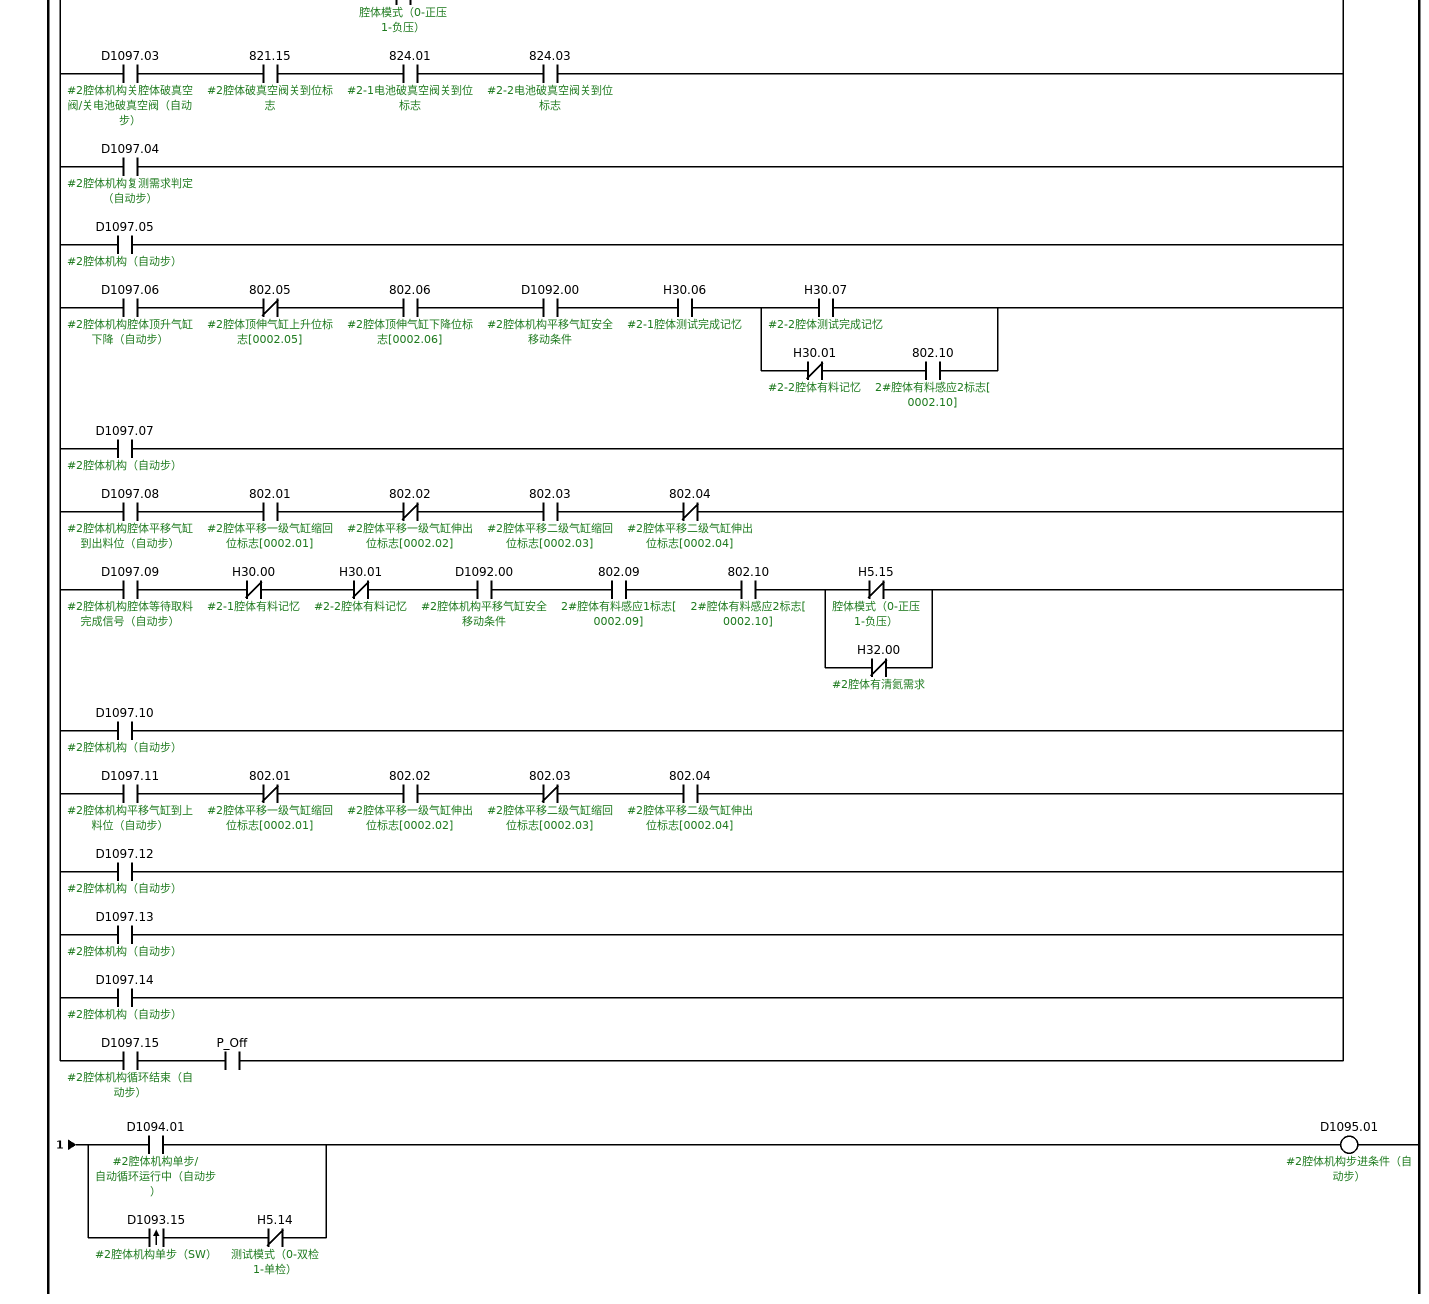
; [picture p264: 氦检机构 / 氦检腔2自动, rungs 7-7]
; rung 7: #2腔体机构步进条件（自动步）
LD D1096.00  ; #2腔体机构自动开始（自动步）
AND T1550  ; #2腔体机构开始运行条件延时(自动步)
LD D1096.01  ; #2腔体机构平移气缸到氦检位/数据初始化（自动步）
ANDNOT 802.01  ; #2腔体平移一级气缸缩回位标志[0002.01]
AND 802.02  ; #2腔体平移一级气缸伸出位标志[0002.02]
AND 802.03  ; #2腔体平移二级气缸缩回位标志[0002.03]
ANDNOT 802.04  ; #2腔体平移二级气缸伸出位标志[0002.04]
AND T1551  ; #2腔体机构数据初始化延时（自动步）
ORLD
LD D1096.02  ; #2腔体机构腔体顶升气缸上升（自动步）
AND 802.05  ; #2腔体顶伸气缸上升位标志[0002.05]
ANDNOT 802.06  ; #2腔体顶伸气缸下降位标志[0002.06]
ORLD
LD D1096.03  ; #2腔体机构等待氦检阀打开条件及腔体抽气阀打开条件/开腔体阀（自动步）
ANDNOT H27.00  ; #1腔体有清氦需求
LDNOT H37.00  ; #3腔体有清氦需求
ANDNOT H47.00  ; #4腔体有清氦需求
ANDNOT H57.00  ; 复检腔体有清氦需求
OR H6.02  ; 加速模式（1-开启）
ANDLD
AND D1092.15  ; #2腔体机构腔体抽气阀打开允许
AND D1092.14  ; #2腔体氦检阀打开允许条件
LD W380.15  ; 氦检仪漏率低于设定值（稳态）
OR H5.02  ; 氦检仪屏蔽
ANDLD
AND=L(301) D1104 #0  ; #2腔体机构清氦步序号
ORLD
OR D1096.04  ; #2腔体机构（自动步）
LD D1096.05  ; #2腔体机构腔体抽气阀打开/延时开电池抽气阀（自动步）
AND T2000  ; #2-1腔体抽真空阈值到达延时（测试）
ANDNOT H31.04  ; #2-1腔体抽真空NG
ANDNOT H31.05  ; #2-2腔体抽真空NG
LD 823.08  ; #2-1电池抽真空阀开到位标志
AND T2020  ; #2-1电池抽真空阈值到达延时（测试）
ANDNOT H31.00  ; #2-1电池泄漏
LD T2320  ; #2-2电池抽真空阈值到达延时（测试）
AND 823.10  ; #2-2电池抽真空阀开到位标志
ANDNOT H31.01  ; #2-2电池泄漏
ORNOT H30.01  ; #2-2腔体有料记忆
ANDLD
OR H5.15  ; 腔体模式（0-正压 1-负压）
OR H5.10  ; 空跑程序
ANDLD
ORLD
LD D1096.06  ; #2腔体机构关电池抽气阀（自动步）
ANDNOT W432.12  ; 设备氦气压力信号#1[alm]
ANDNOT W432.14  ; 设备注氦压力调节阀#1[alm]
AND 823.09  ; #2-1电池抽真空阀关到位标志
AND 823.11  ; #2-2电池抽真空阀关到位标志
ORLD
LD D1096.07  ; #2腔体机构开电池注氦阀（自动步）
LD 823.12  ; #2-1电池注氦阀开到位标志
AND T2024  ; #2-1电池注氦压力到达延时（测试）
LD 823.14  ; #2-2电池注氦阀开到位标志
AND T2324  ; #2-2电池注氦压力到达延时（测试）
ORNOT H30.01  ; #2-2腔体有料记忆
ANDLD
OR H31.02  ; #2-1电池注氦超时
OR H31.03  ; #2-2电池注氦超时
OR H5.15  ; 腔体模式（0-正压 1-负压）
OR H5.10  ; 空跑程序
ANDLD
ORLD
LD D1096.08  ; #2腔体机构关电池注氦阀（自动步）
AND 823.13  ; #2-1电池注氦阀关到位标志
AND 823.15  ; #2-2电池注氦阀关到位标志
ANDNOT H31.02  ; #2-1电池注氦超时
ANDNOT H31.03  ; #2-2电池注氦超时
LDNOT H31.08  ; #2-1注氦超限
ANDNOT H31.09  ; #2-2注氦超限
ORNOT H6.08  ; 注氦超限判断启用（1-启用）
ANDLD
ORLD
OR D1096.09  ; #2腔体机构（自动步）
LD D1096.10  ; #2腔体机构开腔体氦检阀/延时关腔体抽气阀（自动步）
LD T2006  ; #2-1腔体氦检数据取值判定延时（测试）
LD 820.10  ; 清氦保护阀1开到位标志[0000.10]
AND 802.07  ; #2腔体氦检阀开到位标志[0002.07]
OR H5.02  ; 氦检仪屏蔽
ANDLD
LD H31.06  ; #2-1腔体氦检时腔体压力过高
AND H31.07  ; #2-2腔体氦检时腔体压力过高
ORLD
ANDLD
ORLD
OR D1096.11  ; #2腔体机构（自动步）
LD D1096.12  ; #2腔体机构关腔体氦检阀（自动步）
AND 802.08  ; #2腔体氦检阀关到位标志[0002.08]
ANDNOT 802.07  ; #2腔体氦检阀开到位标志[0002.07]
LD 820.11  ; 清氦保护阀1阀关到位标志[0000.11]
ORNOT H6.07  ; 氦检完成后关闭氦检保护阀（1-氦检后关闭）
ANDLD
ORLD
OR D1096.13  ; #2腔体机构（自动步）
LD D1096.14  ; #2腔体机构开腔体#2-1腔体阀/开腔体#2-2腔体阀（自动步）
AND 802.08  ; #2腔体氦检阀关到位标志[0002.08]
ANDNOT H5.15  ; 腔体模式（0-正压 1-负压）
AND D1092.15  ; #2腔体机构腔体抽气阀打开允许
ORLD
LD D1096.15  ; #2腔体机构开腔体抽真空阀/开电池抽真空阀（自动步）
LD T2007  ; #2-1腔体抽残气压力到达延时（测试）
OR T2008  ; #2-1腔体抽残气时间上限到达延时（测试）
ANDLD
LD T2026  ; #2-1电池抽残气压力到达延时（测试）
OR T2027  ; #2-1电池抽残气时间上限到达延时（测试）
LD T2326  ; #2-2电池抽残气压力到达延时（测试）
OR T2327  ; #2-2电池抽残气时间上限到达延时（测试）
ANDLD
OR H5.10  ; 空跑程序
ANDLD
ORLD
LD D1097.00  ; #2腔体机构关腔体抽真空阀/关电池抽真空阀/开腔体阀（自动步）
AND 821.09  ; #2腔体抽真空阀关到位标志
AND 823.09  ; #2-1电池抽真空阀关到位标志
AND 823.11  ; #2-2电池抽真空阀关到位标志
ORLD
LD D1097.01  ; #2腔体机构清氦需求判定（自动步）
LDNOT H32.00  ; #2腔体有清氦需求
OR H5.15  ; 腔体模式（0-正压 1-负压）
ANDLD
ORLD
LD D1097.02  ; #2腔体机构开腔体破真空阀/开电池破真空阀（自动步）
AND T2002  ; #2-1腔体破真空阈值到达延时（测试）
LD T2022  ; #2-1电池破真空阈值到达延时（测试）
AND T2322  ; #2-2电池破真空阈值到达延时（测试）
OR H5.15  ; 腔体模式（0-正压 1-负压）
ANDLD
ORLD
LD D1097.03  ; #2腔体机构关腔体破真空阀/关电池破真空阀（自动步）
AND 821.15  ; #2腔体破真空阀关到位标志
AND 824.01  ; #2-1电池破真空阀关到位标志
AND 824.03  ; #2-2电池破真空阀关到位标志
ORLD
OR D1097.04  ; #2腔体机构复测需求判定（自动步）
OR D1097.05  ; #2腔体机构（自动步）
LD D1097.06  ; #2腔体机构腔体顶升气缸下降（自动步）
ANDNOT 802.05  ; #2腔体顶伸气缸上升位标志[0002.05]
AND 802.06  ; #2腔体顶伸气缸下降位标志[0002.06]
AND D1092.00  ; #2腔体机构平移气缸安全移动条件
AND H30.06  ; #2-1腔体测试完成记忆
LD H30.07  ; #2-2腔体测试完成记忆
LDNOT H30.01  ; #2-2腔体有料记忆
AND 802.10  ; 2#腔体有料感应2标志[0002.10]
ORLD
ANDLD
ORLD
OR D1097.07  ; #2腔体机构（自动步）
LD D1097.08  ; #2腔体机构腔体平移气缸到出料位（自动步）
AND 802.01  ; #2腔体平移一级气缸缩回位标志[0002.01]
ANDNOT 802.02  ; #2腔体平移一级气缸伸出位标志[0002.02]
AND 802.03  ; #2腔体平移二级气缸缩回位标志[0002.03]
ANDNOT 802.04  ; #2腔体平移二级气缸伸出位标志[0002.04]
ORLD
LD D1097.09  ; #2腔体机构腔体等待取料完成信号（自动步）  // 负压有清氦需求时，无需回初始位,直接跳回初始步序（D1096.00）
ANDNOT H30.00  ; #2-1腔体有料记忆
ANDNOT H30.01  ; #2-2腔体有料记忆
AND D1092.00  ; #2腔体机构平移气缸安全移动条件
AND 802.09  ; 2#腔体有料感应1标志[0002.09]
AND 802.10  ; 2#腔体有料感应2标志[0002.10]
LDNOT H5.15  ; 腔体模式（0-正压 1-负压）
ORNOT H32.00  ; #2腔体有清氦需求
ANDLD
ORLD
OR D1097.10  ; #2腔体机构（自动步）
LD D1097.11  ; #2腔体机构平移气缸到上料位（自动步）
ANDNOT 802.01  ; #2腔体平移一级气缸缩回位标志[0002.01]
AND 802.02  ; #2腔体平移一级气缸伸出位标志[0002.02]
ANDNOT 802.03  ; #2腔体平移二级气缸缩回位标志[0002.03]
AND 802.04  ; #2腔体平移二级气缸伸出位标志[0002.04]
ORLD
OR D1097.12  ; #2腔体机构（自动步）
OR D1097.13  ; #2腔体机构（自动步）
OR D1097.14  ; #2腔体机构（自动步）
LD D1097.15  ; #2腔体机构循环结束（自动步）
AND P_Off
ORLD
LD D1094.01  ; #2腔体机构单步/自动循环运行中（自动步）
@LD D1093.15  ; #2腔体机构单步（SW）
ANDNOT H5.14  ; 测试模式（0-双检 1-单检）
ORLD
ANDLD
OUT D1095.01  ; #2腔体机构步进条件（自动步）

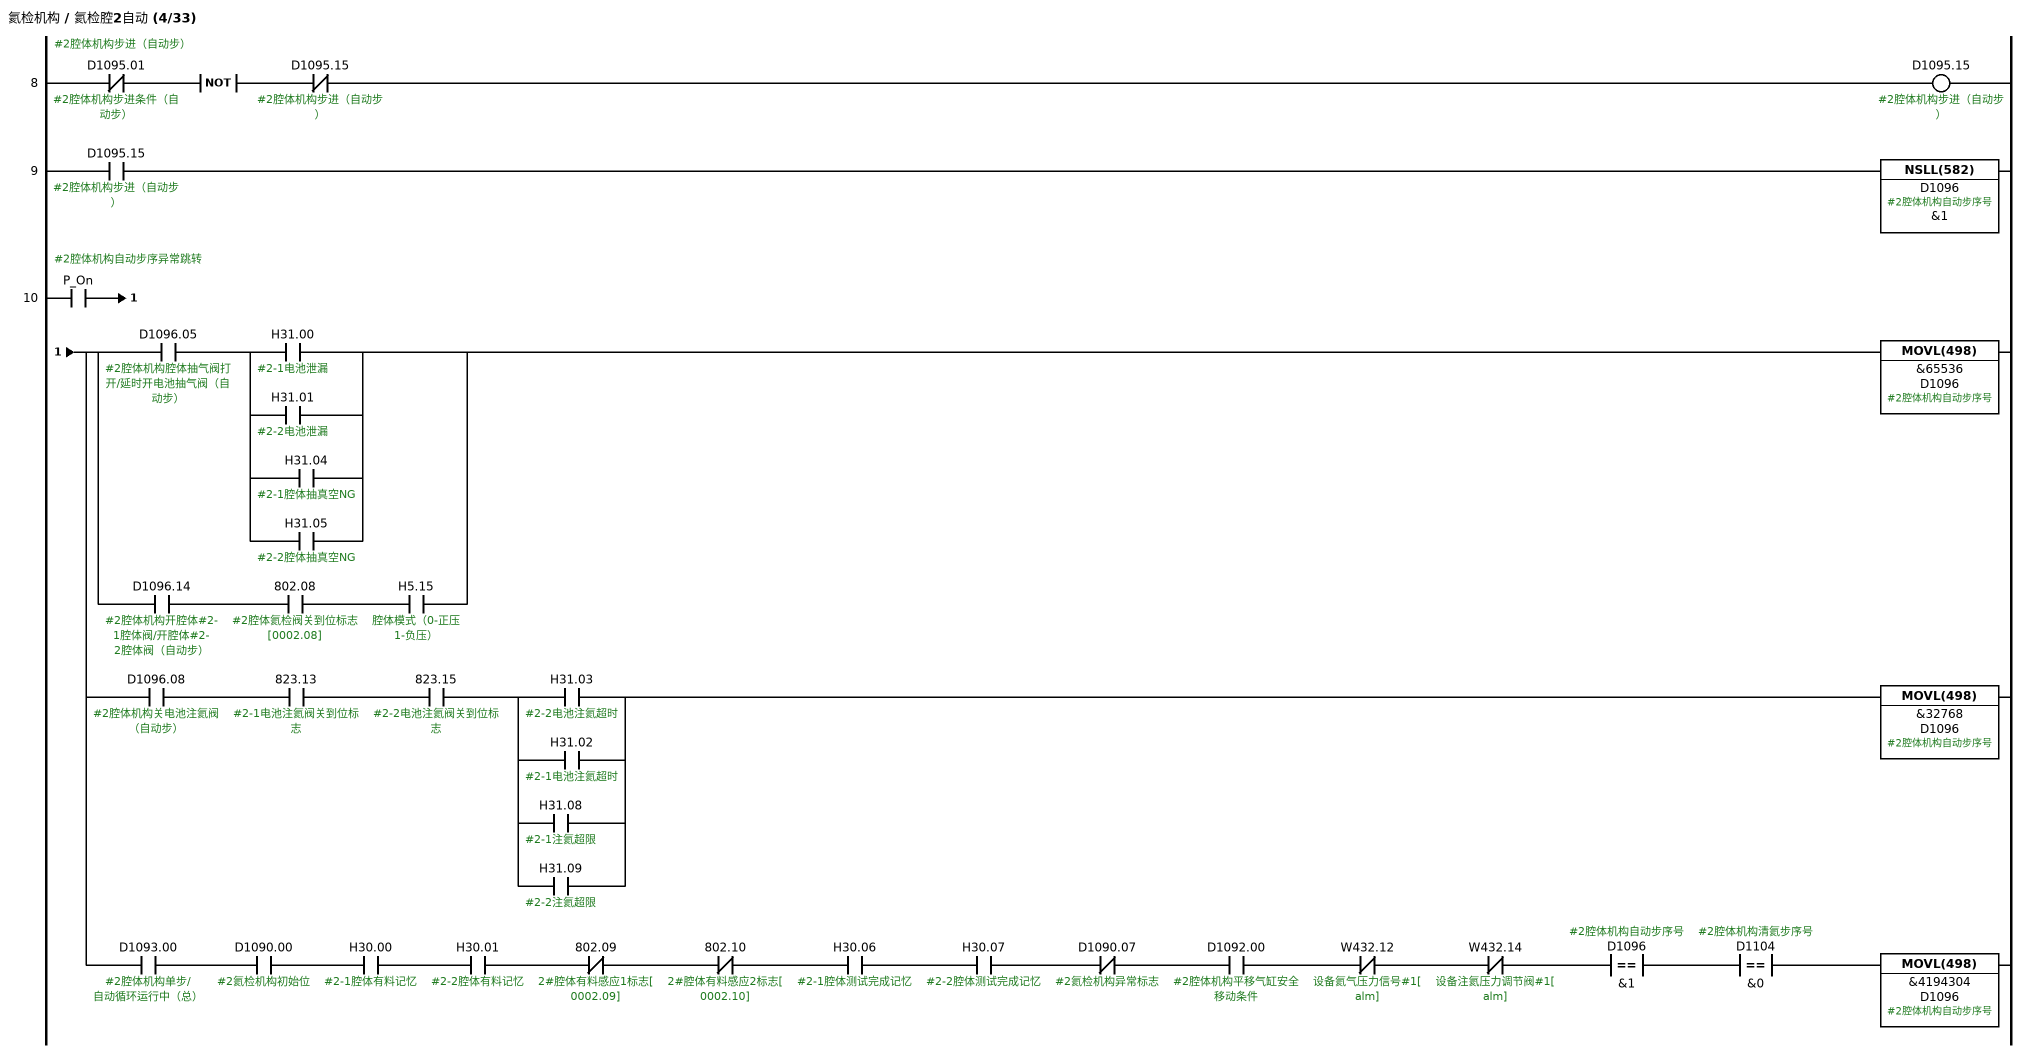
; rung 8: #2腔体机构步进（自动步）
LDNOT D1095.01  ; #2腔体机构步进条件（自动步）
NOT(520)
ANDNOT D1095.15  ; #2腔体机构步进（自动步）
OUT D1095.15  ; #2腔体机构步进（自动步）
; rung 9
LD D1095.15  ; #2腔体机构步进（自动步）
NSLL(582) D1096 &1  ; #2腔体机构自动步序号
; rung 10: #2腔体机构自动步序异常跳转
LD P_On
OUT TR0
LD D1096.05  ; #2腔体机构腔体抽气阀打开/延时开电池抽气阀（自动步）
LD H31.00  ; #2-1电池泄漏
OR H31.01  ; #2-2电池泄漏
OR H31.04  ; #2-1腔体抽真空NG
OR H31.05  ; #2-2腔体抽真空NG
ANDLD
LD D1096.14  ; #2腔体机构开腔体#2-1腔体阀/开腔体#2-2腔体阀（自动步）  // 负压模式不需要进行氦检后抽真空动作
AND 802.08  ; #2腔体氦检阀关到位标志[0002.08]
AND H5.15  ; 腔体模式（0-正压 1-负压）
ORLD
ANDLD
MOVL(498) &65536 D1096  ; #2腔体机构自动步序号  // 出现腔体抽真空NG，双电池抽真空NG，均跳转至自动步序D1067.0
LD TR0
AND D1096.08  ; #2腔体机构关电池注氦阀（自动步）
AND 823.13  ; #2-1电池注氦阀关到位标志
AND 823.15  ; #2-2电池注氦阀关到位标志
LD H31.03  ; #2-2电池注氦超时
OR H31.02  ; #2-1电池注氦超时
OR H31.08  ; #2-1注氦超限
OR H31.09  ; #2-2注氦超限
ANDLD
MOVL(498) &32768 D1096  ; #2腔体机构自动步序号
LD TR0
AND D1093.00  ; #2腔体机构单步/自动循环运行中（总）
AND D1090.00  ; #2氦检机构初始位
AND H30.00  ; #2-1腔体有料记忆
AND H30.01  ; #2-2腔体有料记忆
ANDNOT 802.09  ; 2#腔体有料感应1标志[0002.09]
ANDNOT 802.10  ; 2#腔体有料感应2标志[0002.10]
AND H30.06  ; #2-1腔体测试完成记忆
AND H30.07  ; #2-2腔体测试完成记忆
ANDNOT D1090.07  ; #2氦检机构异常标志
AND D1092.00  ; #2腔体机构平移气缸安全移动条件
ANDNOT W432.12  ; 设备氦气压力信号#1[alm]
ANDNOT W432.14  ; 设备注氦压力调节阀#1[alm]
AND=L(301) D1096 &1  ; #2腔体机构自动步序号
AND=L(301) D1104 &0  ; #2腔体机构清氦步序号
MOVL(498) &4194304 D1096  ; #2腔体机构自动步序号  // 带料复位，有测试完成物料跳转至D1097.06
; rung 11: ******************************* / 清氦步序 / *******************************

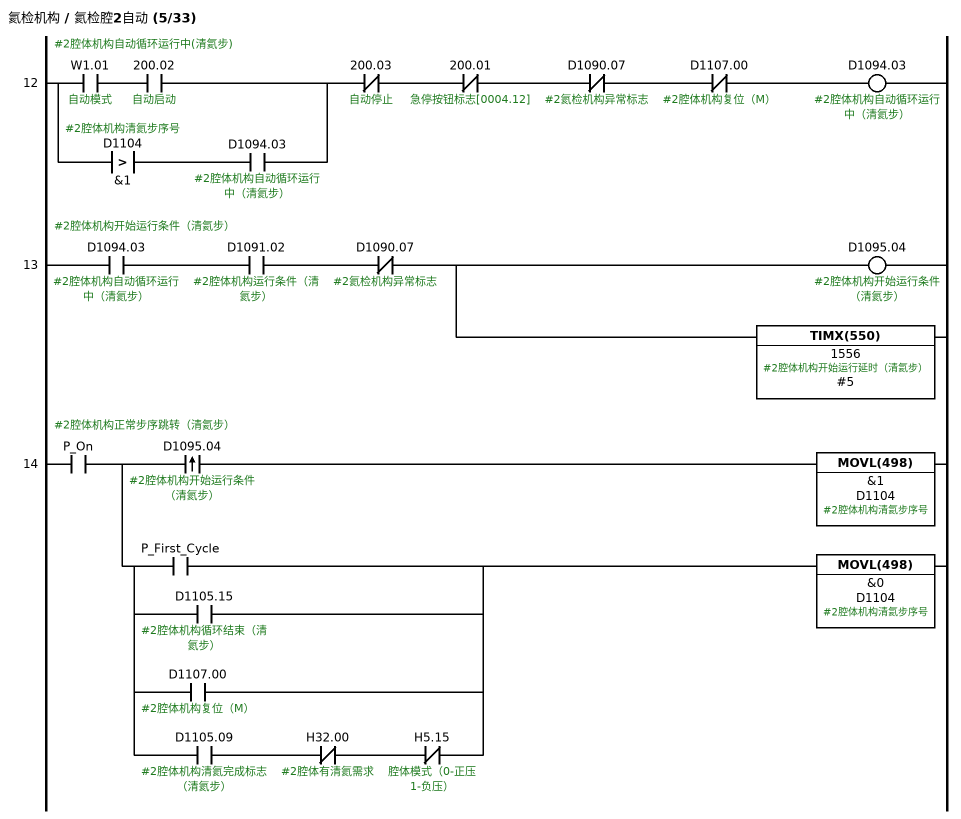
; rung 12: #2腔体机构自动循环运行中(清氦步)
LD W1.01  ; 自动模式
AND 200.02  ; 自动启动
LD>L(321) D1104 &1  ; #2腔体机构清氦步序号
AND D1094.03  ; #2腔体机构自动循环运行中（清氦步）
ORLD
ANDNOT 200.03  ; 自动停止
ANDNOT 200.01  ; 急停按钮标志[0004.12]
ANDNOT D1090.07  ; #2氦检机构异常标志
ANDNOT D1107.00  ; #2腔体机构复位（M）
OUT D1094.03  ; #2腔体机构自动循环运行中（清氦步）
; rung 13: #2腔体机构开始运行条件（清氦步）
LD D1094.03  ; #2腔体机构自动循环运行中（清氦步）
AND D1091.02  ; #2腔体机构运行条件（清氦步）
ANDNOT D1090.07  ; #2氦检机构异常标志
OUT D1095.04  ; #2腔体机构开始运行条件（清氦步）
TIMX(550) 1556 #5  ; #2腔体机构开始运行延时（清氦步）
; rung 14: #2腔体机构正常步序跳转（清氦步）
LD P_On
OUT TR0
@AND D1095.04  ; #2腔体机构开始运行条件（清氦步）
MOVL(498) &1 D1104  ; #2腔体机构清氦步序号
LD TR0
LD P_First_Cycle
OR D1105.15  ; #2腔体机构循环结束（清氦步）
OR D1107.00  ; #2腔体机构复位（M）
LD D1105.09  ; #2腔体机构清氦完成标志（清氦步）  // 正压腔体是待料清氦，需跳转回测试步序
ANDNOT H32.00  ; #2腔体有清氦需求
ANDNOT H5.15  ; 腔体模式（0-正压 1-负压）
ORLD
ANDLD
MOVL(498) &0 D1104  ; #2腔体机构清氦步序号

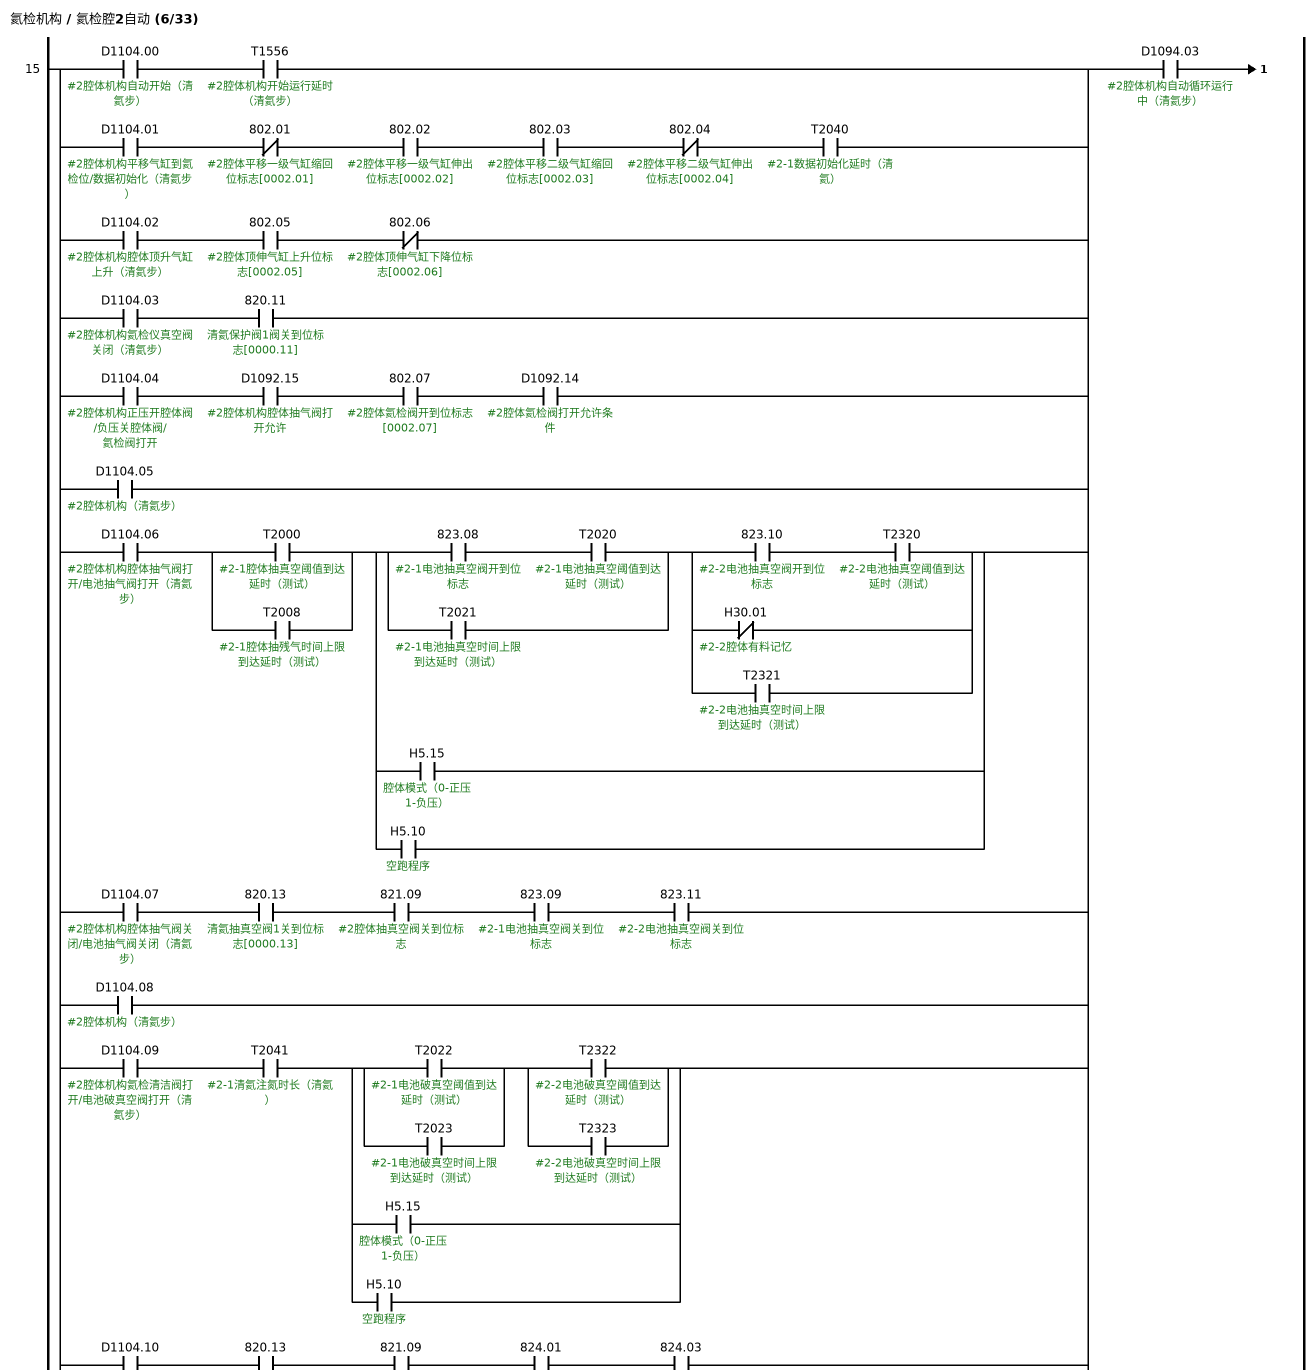

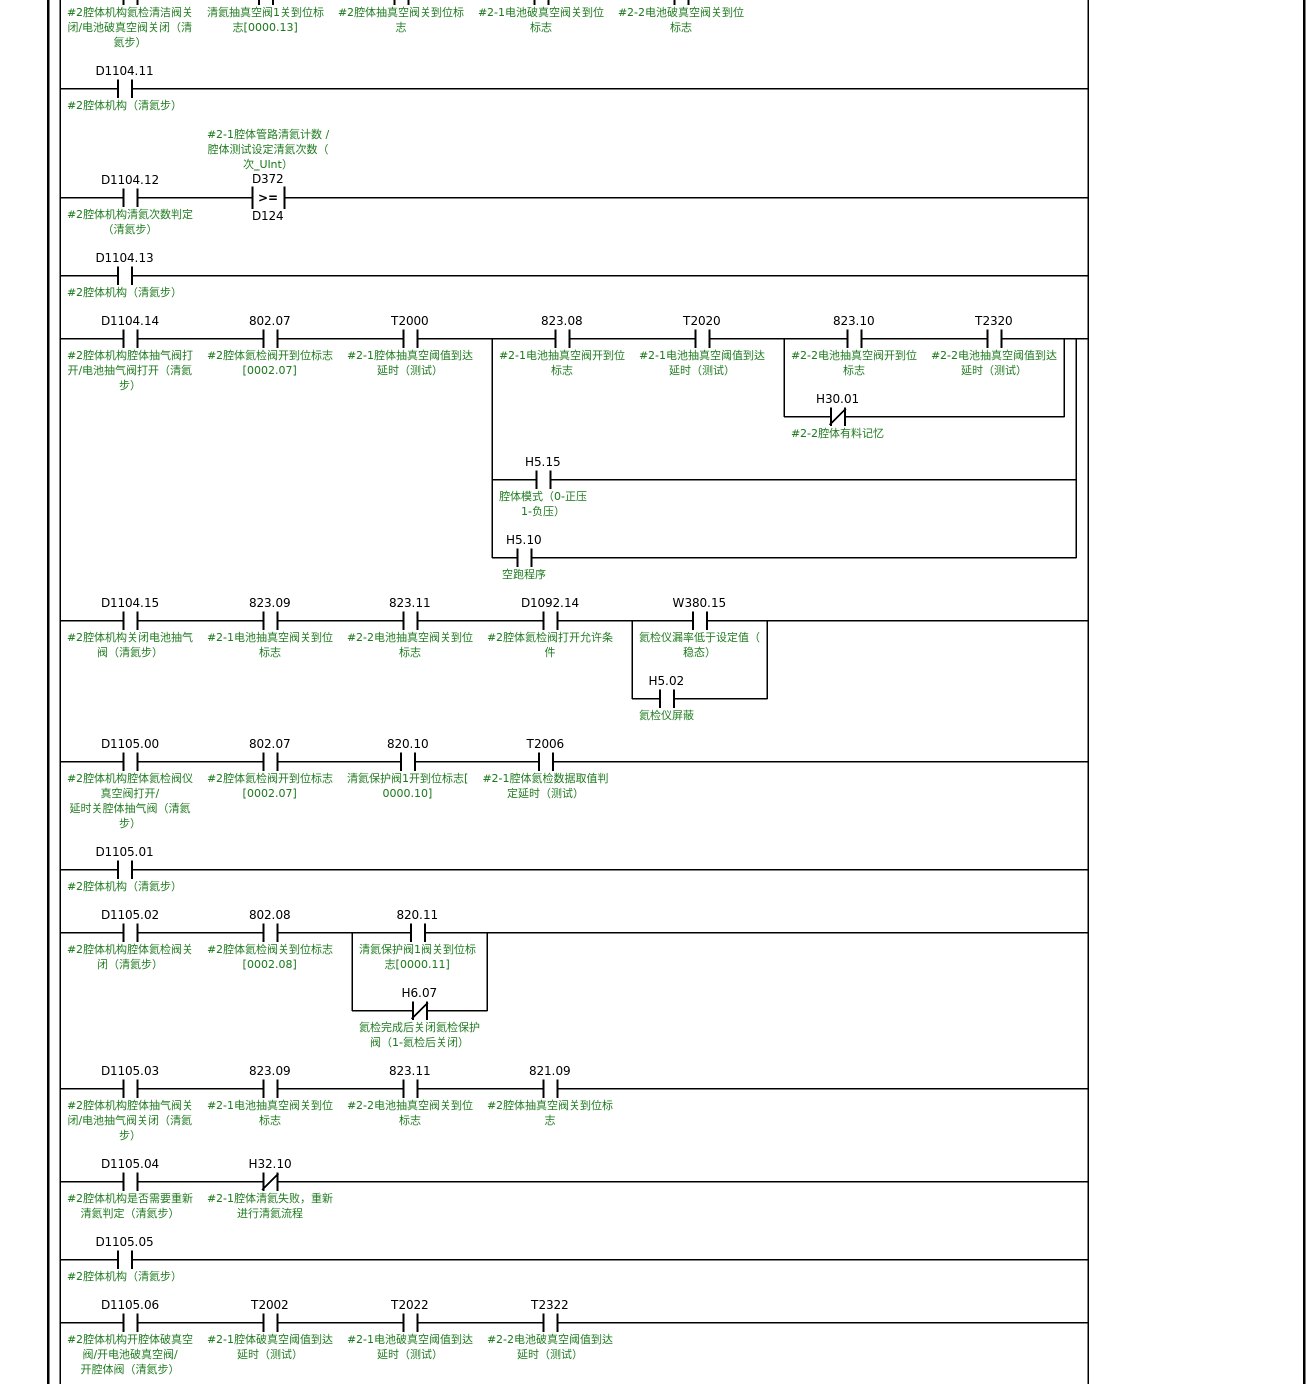

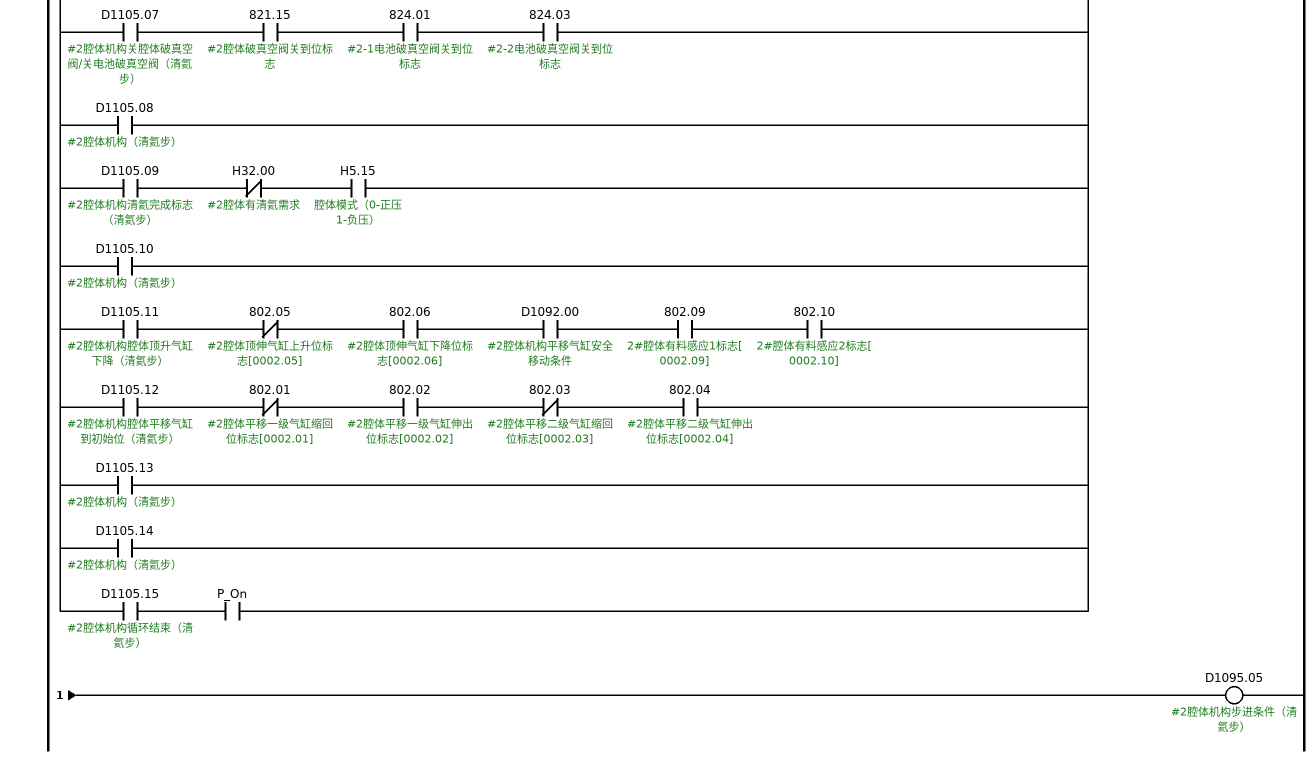
; rung 15
LD D1104.00  ; #2腔体机构自动开始（清氦步）
AND T1556  ; #2腔体机构开始运行延时（清氦步）
LD D1104.01  ; #2腔体机构平移气缸到氦检位/数据初始化（清氦步）
ANDNOT 802.01  ; #2腔体平移一级气缸缩回位标志[0002.01]
AND 802.02  ; #2腔体平移一级气缸伸出位标志[0002.02]
AND 802.03  ; #2腔体平移二级气缸缩回位标志[0002.03]
ANDNOT 802.04  ; #2腔体平移二级气缸伸出位标志[0002.04]
AND T2040  ; #2-1数据初始化延时（清氦）
ORLD
LD D1104.02  ; #2腔体机构腔体顶升气缸上升（清氦步）
AND 802.05  ; #2腔体顶伸气缸上升位标志[0002.05]
ANDNOT 802.06  ; #2腔体顶伸气缸下降位标志[0002.06]
ORLD
LD D1104.03  ; #2腔体机构氦检仪真空阀关闭（清氦步）
AND 820.11  ; 清氦保护阀1阀关到位标志[0000.11]
ORLD
LD D1104.04  ; #2腔体机构正压开腔体阀/负压关腔体阀/氦检阀打开  // 负压模式下，复测前的清氦不允许抽电池
AND D1092.15  ; #2腔体机构腔体抽气阀打开允许
AND 802.07  ; #2腔体氦检阀开到位标志[0002.07]
AND D1092.14  ; #2腔体氦检阀打开允许条件
ORLD
OR D1104.05  ; #2腔体机构（清氦步）
LD D1104.06  ; #2腔体机构腔体抽气阀打开/电池抽气阀打开（清氦步）
LD T2000  ; #2-1腔体抽真空阈值到达延时（测试）
OR T2008  ; #2-1腔体抽残气时间上限到达延时（测试）
ANDLD
LD 823.08  ; #2-1电池抽真空阀开到位标志
AND T2020  ; #2-1电池抽真空阈值到达延时（测试）
OR T2021  ; #2-1电池抽真空时间上限到达延时（测试）
LD 823.10  ; #2-2电池抽真空阀开到位标志
AND T2320  ; #2-2电池抽真空阈值到达延时（测试）
ORNOT H30.01  ; #2-2腔体有料记忆
OR T2321  ; #2-2电池抽真空时间上限到达延时（测试）
ANDLD
OR H5.15  ; 腔体模式（0-正压 1-负压）
OR H5.10  ; 空跑程序
ANDLD
ORLD
LD D1104.07  ; #2腔体机构腔体抽气阀关闭/电池抽气阀关闭（清氦步）
AND 820.13  ; 清氦抽真空阀1关到位标志[0000.13]
AND 821.09  ; #2腔体抽真空阀关到位标志
AND 823.09  ; #2-1电池抽真空阀关到位标志
AND 823.11  ; #2-2电池抽真空阀关到位标志
ORLD
OR D1104.08  ; #2腔体机构（清氦步）
LD D1104.09  ; #2腔体机构氦检清洁阀打开/电池破真空阀打开（清氦步）
AND T2041  ; #2-1清氦注氮时长（清氦）
LD T2022  ; #2-1电池破真空阈值到达延时（测试）
OR T2023  ; #2-1电池破真空时间上限到达延时（测试）
LD T2322  ; #2-2电池破真空阈值到达延时（测试）
OR T2323  ; #2-2电池破真空时间上限到达延时（测试）
ANDLD
OR H5.15  ; 腔体模式（0-正压 1-负压）
OR H5.10  ; 空跑程序
ANDLD
ORLD
LD D1104.10  ; #2腔体机构氦检清洁阀关闭/电池破真空阀关闭（清氦步）
AND 820.13  ; 清氦抽真空阀1关到位标志[0000.13]
AND 821.09  ; #2腔体抽真空阀关到位标志
AND 824.01  ; #2-1电池破真空阀关到位标志
AND 824.03  ; #2-2电池破真空阀关到位标志
ORLD
OR D1104.11  ; #2腔体机构（清氦步）
LD D1104.12  ; #2腔体机构清氦次数判定（清氦步）
AND>=(325) D372 D124  ; #2-1腔体管路清氦计数, 腔体测试设定清氦次数（次_UInt）
ORLD
OR D1104.13  ; #2腔体机构（清氦步）
LD D1104.14  ; #2腔体机构腔体抽气阀打开/电池抽气阀打开（清氦步）
AND 802.07  ; #2腔体氦检阀开到位标志[0002.07]
AND T2000  ; #2-1腔体抽真空阈值到达延时（测试）
LD 823.08  ; #2-1电池抽真空阀开到位标志
AND T2020  ; #2-1电池抽真空阈值到达延时（测试）
LD 823.10  ; #2-2电池抽真空阀开到位标志
AND T2320  ; #2-2电池抽真空阈值到达延时（测试）
ORNOT H30.01  ; #2-2腔体有料记忆
ANDLD
OR H5.15  ; 腔体模式（0-正压 1-负压）
OR H5.10  ; 空跑程序
ANDLD
ORLD
LD D1104.15  ; #2腔体机构关闭电池抽气阀（清氦步）
AND 823.09  ; #2-1电池抽真空阀关到位标志
AND 823.11  ; #2-2电池抽真空阀关到位标志
AND D1092.14  ; #2腔体氦检阀打开允许条件
LD W380.15  ; 氦检仪漏率低于设定值（稳态）
OR H5.02  ; 氦检仪屏蔽
ANDLD
ORLD
LD D1105.00  ; #2腔体机构腔体氦检阀仪真空阀打开/延时关腔体抽气阀（清氦步）
AND 802.07  ; #2腔体氦检阀开到位标志[0002.07]
AND 820.10  ; 清氦保护阀1开到位标志[0000.10]
AND T2006  ; #2-1腔体氦检数据取值判定延时（测试）
ORLD
OR D1105.01  ; #2腔体机构（清氦步）
LD D1105.02  ; #2腔体机构腔体氦检阀关闭（清氦步）
AND 802.08  ; #2腔体氦检阀关到位标志[0002.08]
LD 820.11  ; 清氦保护阀1阀关到位标志[0000.11]
ORNOT H6.07  ; 氦检完成后关闭氦检保护阀（1-氦检后关闭）
ANDLD
ORLD
LD D1105.03  ; #2腔体机构腔体抽气阀关闭/电池抽气阀关闭（清氦步）
AND 823.09  ; #2-1电池抽真空阀关到位标志
AND 823.11  ; #2-2电池抽真空阀关到位标志
AND 821.09  ; #2腔体抽真空阀关到位标志
ORLD
LD D1105.04  ; #2腔体机构是否需要重新清氦判定（清氦步）
ANDNOT H32.10  ; #2-1腔体清氦失败，重新进行清氦流程  // 清氦失败，重新进行清氦
ORLD
OR D1105.05  ; #2腔体机构（清氦步）
LD D1105.06  ; #2腔体机构开腔体破真空阀/开电池破真空阀/开腔体阀（清氦步）
AND T2002  ; #2-1腔体破真空阈值到达延时（测试）
AND T2022  ; #2-1电池破真空阈值到达延时（测试）
AND T2322  ; #2-2电池破真空阈值到达延时（测试）
ORLD
LD D1105.07  ; #2腔体机构关腔体破真空阀/关电池破真空阀（清氦步）
AND 821.15  ; #2腔体破真空阀关到位标志
AND 824.01  ; #2-1电池破真空阀关到位标志
AND 824.03  ; #2-2电池破真空阀关到位标志
ORLD
OR D1105.08  ; #2腔体机构（清氦步）
LD D1105.09  ; #2腔体机构清氦完成标志（清氦步）  // 正压腔体是待料清氦，需跳转回测试步序
ANDNOT H32.00  ; #2腔体有清氦需求
AND H5.15  ; 腔体模式（0-正压 1-负压）
ORLD
OR D1105.10  ; #2腔体机构（清氦步）
LD D1105.11  ; #2腔体机构腔体顶升气缸下降（清氦步）
ANDNOT 802.05  ; #2腔体顶伸气缸上升位标志[0002.05]
AND 802.06  ; #2腔体顶伸气缸下降位标志[0002.06]
AND D1092.00  ; #2腔体机构平移气缸安全移动条件
AND 802.09  ; 2#腔体有料感应1标志[0002.09]
AND 802.10  ; 2#腔体有料感应2标志[0002.10]
ORLD
LD D1105.12  ; #2腔体机构腔体平移气缸到初始位（清氦步）
ANDNOT 802.01  ; #2腔体平移一级气缸缩回位标志[0002.01]
AND 802.02  ; #2腔体平移一级气缸伸出位标志[0002.02]
ANDNOT 802.03  ; #2腔体平移二级气缸缩回位标志[0002.03]
AND 802.04  ; #2腔体平移二级气缸伸出位标志[0002.04]
ORLD
OR D1105.13  ; #2腔体机构（清氦步）
OR D1105.14  ; #2腔体机构（清氦步）
LD D1105.15  ; #2腔体机构循环结束（清氦步）
AND P_On
ORLD
AND D1094.03  ; #2腔体机构自动循环运行中（清氦步）
OUT D1095.05  ; #2腔体机构步进条件（清氦步）

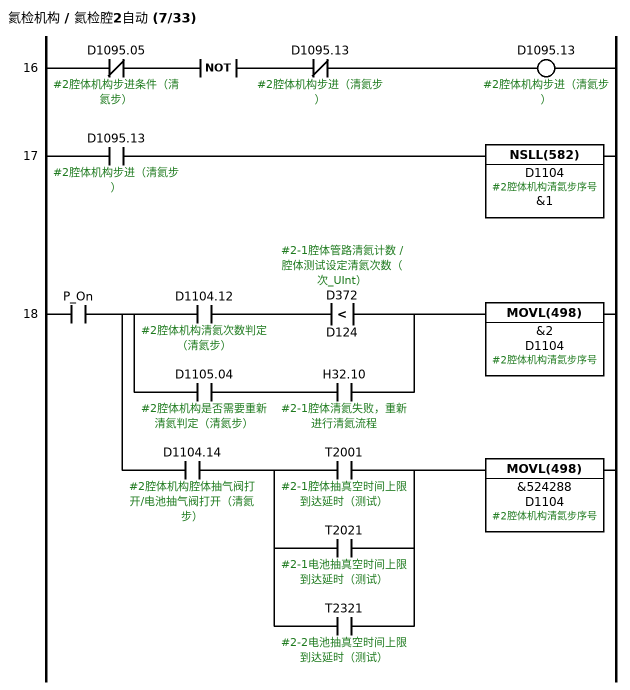
; rung 16
LDNOT D1095.05  ; #2腔体机构步进条件（清氦步）
NOT(520)
ANDNOT D1095.13  ; #2腔体机构步进（清氦步）
OUT D1095.13  ; #2腔体机构步进（清氦步）
; rung 17
LD D1095.13  ; #2腔体机构步进（清氦步）
NSLL(582) D1104 &1  ; #2腔体机构清氦步序号
; rung 18
LD P_On
OUT TR0
LD D1104.12  ; #2腔体机构清氦次数判定（清氦步）
AND<(310) D372 D124  ; #2-1腔体管路清氦计数, 腔体测试设定清氦次数（次_UInt）
LD D1105.04  ; #2腔体机构是否需要重新清氦判定（清氦步）
AND H32.10  ; #2-1腔体清氦失败，重新进行清氦流程  // 清氦失败，重新进行清氦
ORLD
ANDLD
MOVL(498) &2 D1104  ; #2腔体机构清氦步序号
LD TR0
AND D1104.14  ; #2腔体机构腔体抽气阀打开/电池抽气阀打开（清氦步）
LD T2001  ; #2-1腔体抽真空时间上限到达延时（测试）
OR T2021  ; #2-1电池抽真空时间上限到达延时（测试）
OR T2321  ; #2-2电池抽真空时间上限到达延时（测试）
ANDLD
MOVL(498) &524288 D1104  ; #2腔体机构清氦步序号  // 清氦过程腔体或电池抽气上限达到，均直接判定清氦完成，不进入氦检步序（跳转至D1075.03）

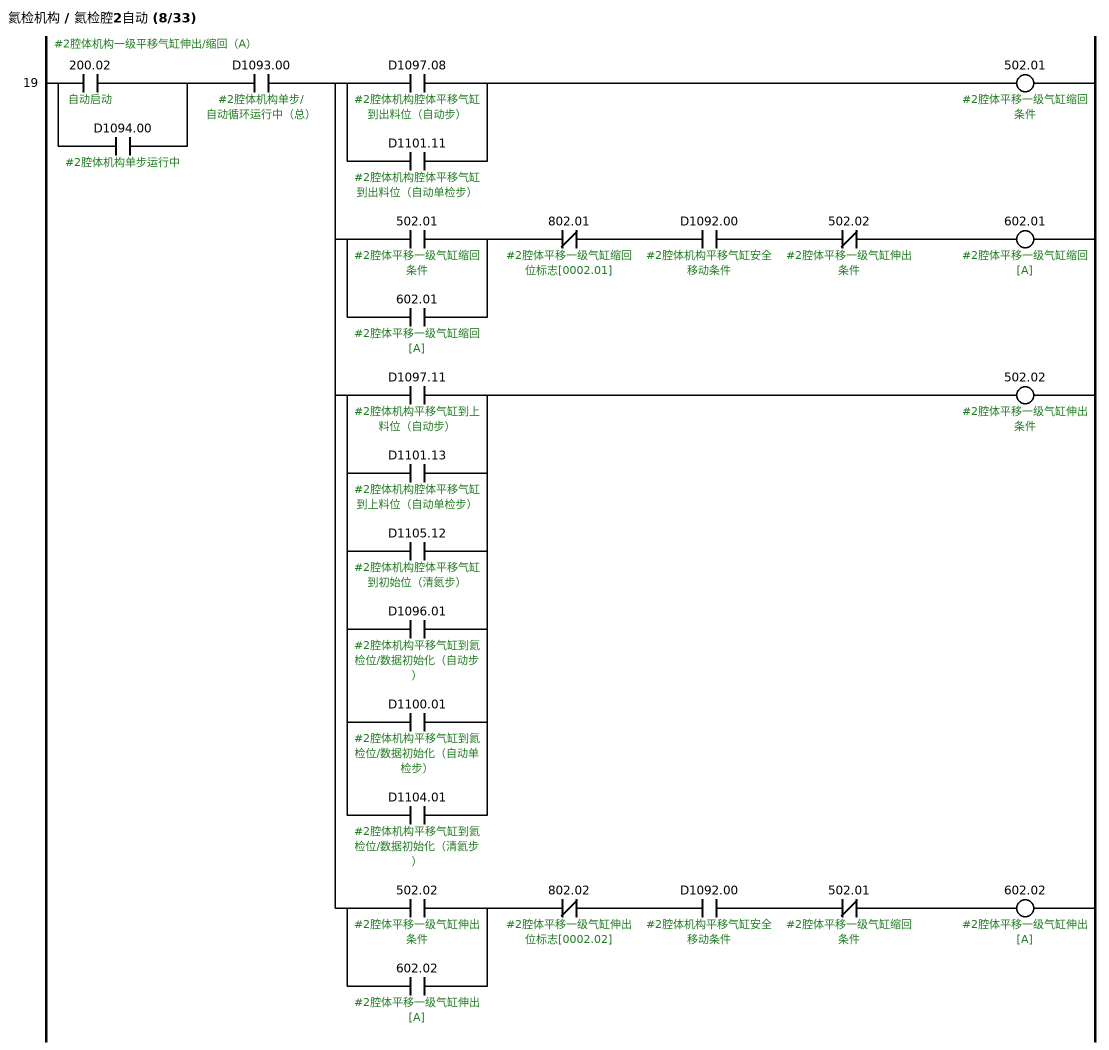
; rung 19: #2腔体机构一级平移气缸伸出/缩回（A）
LD 200.02  ; 自动启动
OR D1094.00  ; #2腔体机构单步运行中
AND D1093.00  ; #2腔体机构单步/自动循环运行中（总）
OUT TR0
LD D1097.08  ; #2腔体机构腔体平移气缸到出料位（自动步）
OR D1101.11  ; #2腔体机构腔体平移气缸到出料位（自动单检步）
ANDLD
OUT 502.01  ; #2腔体平移一级气缸缩回条件
LD TR0
LD 502.01  ; #2腔体平移一级气缸缩回条件
OR 602.01  ; #2腔体平移一级气缸缩回[A]
ANDLD
ANDNOT 802.01  ; #2腔体平移一级气缸缩回位标志[0002.01]
AND D1092.00  ; #2腔体机构平移气缸安全移动条件
ANDNOT 502.02  ; #2腔体平移一级气缸伸出条件
OUT 602.01  ; #2腔体平移一级气缸缩回[A]
LD TR0
LD D1097.11  ; #2腔体机构平移气缸到上料位（自动步）
OR D1101.13  ; #2腔体机构腔体平移气缸到上料位（自动单检步）
OR D1105.12  ; #2腔体机构腔体平移气缸到初始位（清氦步）
OR D1096.01  ; #2腔体机构平移气缸到氦检位/数据初始化（自动步）
OR D1100.01  ; #2腔体机构平移气缸到氦检位/数据初始化（自动单检步）
OR D1104.01  ; #2腔体机构平移气缸到氦检位/数据初始化（清氦步）
ANDLD
OUT 502.02  ; #2腔体平移一级气缸伸出条件
LD TR0
LD 502.02  ; #2腔体平移一级气缸伸出条件
OR 602.02  ; #2腔体平移一级气缸伸出[A]
ANDLD
ANDNOT 802.02  ; #2腔体平移一级气缸伸出位标志[0002.02]
AND D1092.00  ; #2腔体机构平移气缸安全移动条件
ANDNOT 502.01  ; #2腔体平移一级气缸缩回条件
OUT 602.02  ; #2腔体平移一级气缸伸出[A]

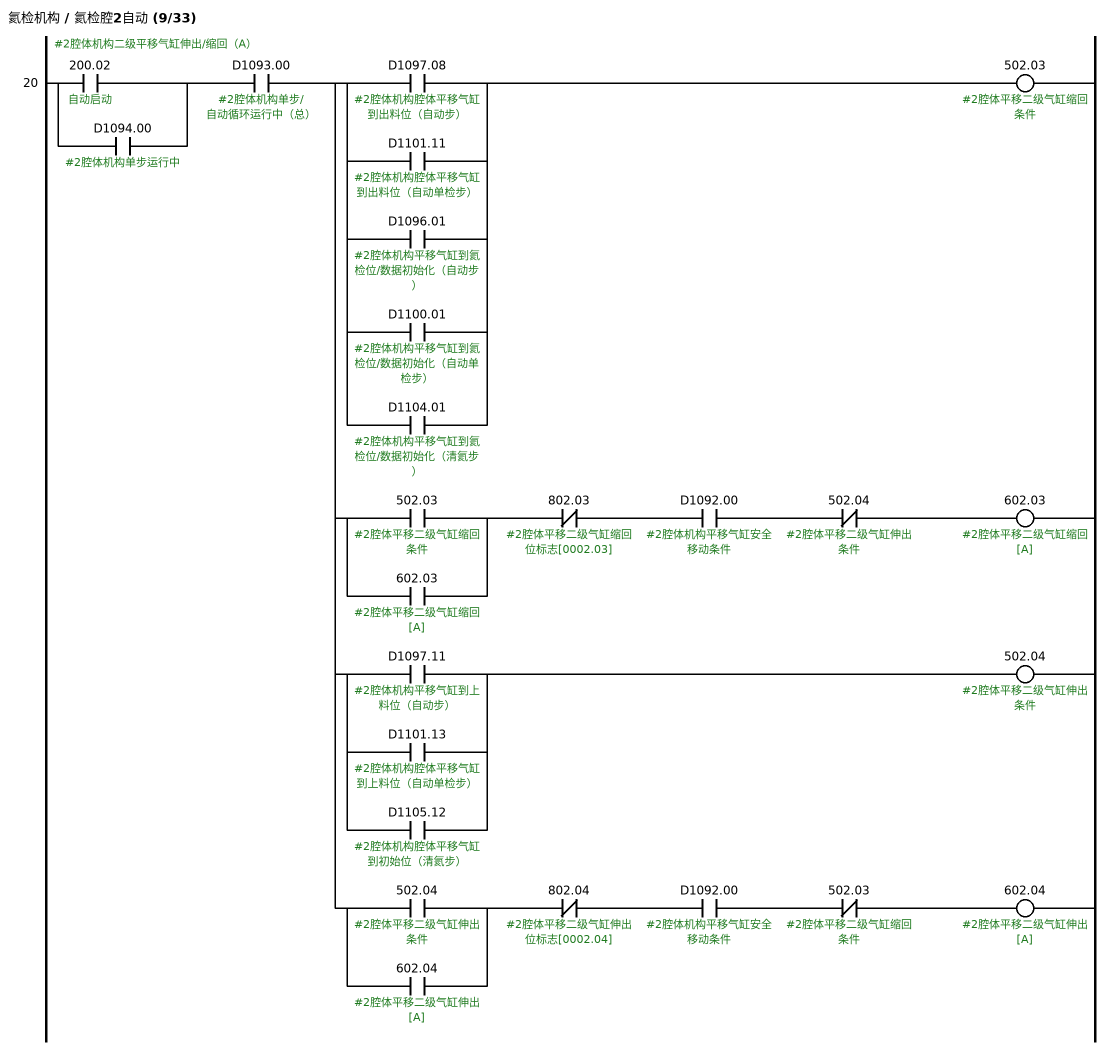
; rung 20: #2腔体机构二级平移气缸伸出/缩回（A）
LD 200.02  ; 自动启动
OR D1094.00  ; #2腔体机构单步运行中
AND D1093.00  ; #2腔体机构单步/自动循环运行中（总）
OUT TR0
LD D1097.08  ; #2腔体机构腔体平移气缸到出料位（自动步）
OR D1101.11  ; #2腔体机构腔体平移气缸到出料位（自动单检步）
OR D1096.01  ; #2腔体机构平移气缸到氦检位/数据初始化（自动步）
OR D1100.01  ; #2腔体机构平移气缸到氦检位/数据初始化（自动单检步）
OR D1104.01  ; #2腔体机构平移气缸到氦检位/数据初始化（清氦步）
ANDLD
OUT 502.03  ; #2腔体平移二级气缸缩回条件
LD TR0
LD 502.03  ; #2腔体平移二级气缸缩回条件
OR 602.03  ; #2腔体平移二级气缸缩回[A]
ANDLD
ANDNOT 802.03  ; #2腔体平移二级气缸缩回位标志[0002.03]
AND D1092.00  ; #2腔体机构平移气缸安全移动条件
ANDNOT 502.04  ; #2腔体平移二级气缸伸出条件
OUT 602.03  ; #2腔体平移二级气缸缩回[A]
LD TR0
LD D1097.11  ; #2腔体机构平移气缸到上料位（自动步）
OR D1101.13  ; #2腔体机构腔体平移气缸到上料位（自动单检步）
OR D1105.12  ; #2腔体机构腔体平移气缸到初始位（清氦步）
ANDLD
OUT 502.04  ; #2腔体平移二级气缸伸出条件
LD TR0
LD 502.04  ; #2腔体平移二级气缸伸出条件
OR 602.04  ; #2腔体平移二级气缸伸出[A]
ANDLD
ANDNOT 802.04  ; #2腔体平移二级气缸伸出位标志[0002.04]
AND D1092.00  ; #2腔体机构平移气缸安全移动条件
ANDNOT 502.03  ; #2腔体平移二级气缸缩回条件
OUT 602.04  ; #2腔体平移二级气缸伸出[A]

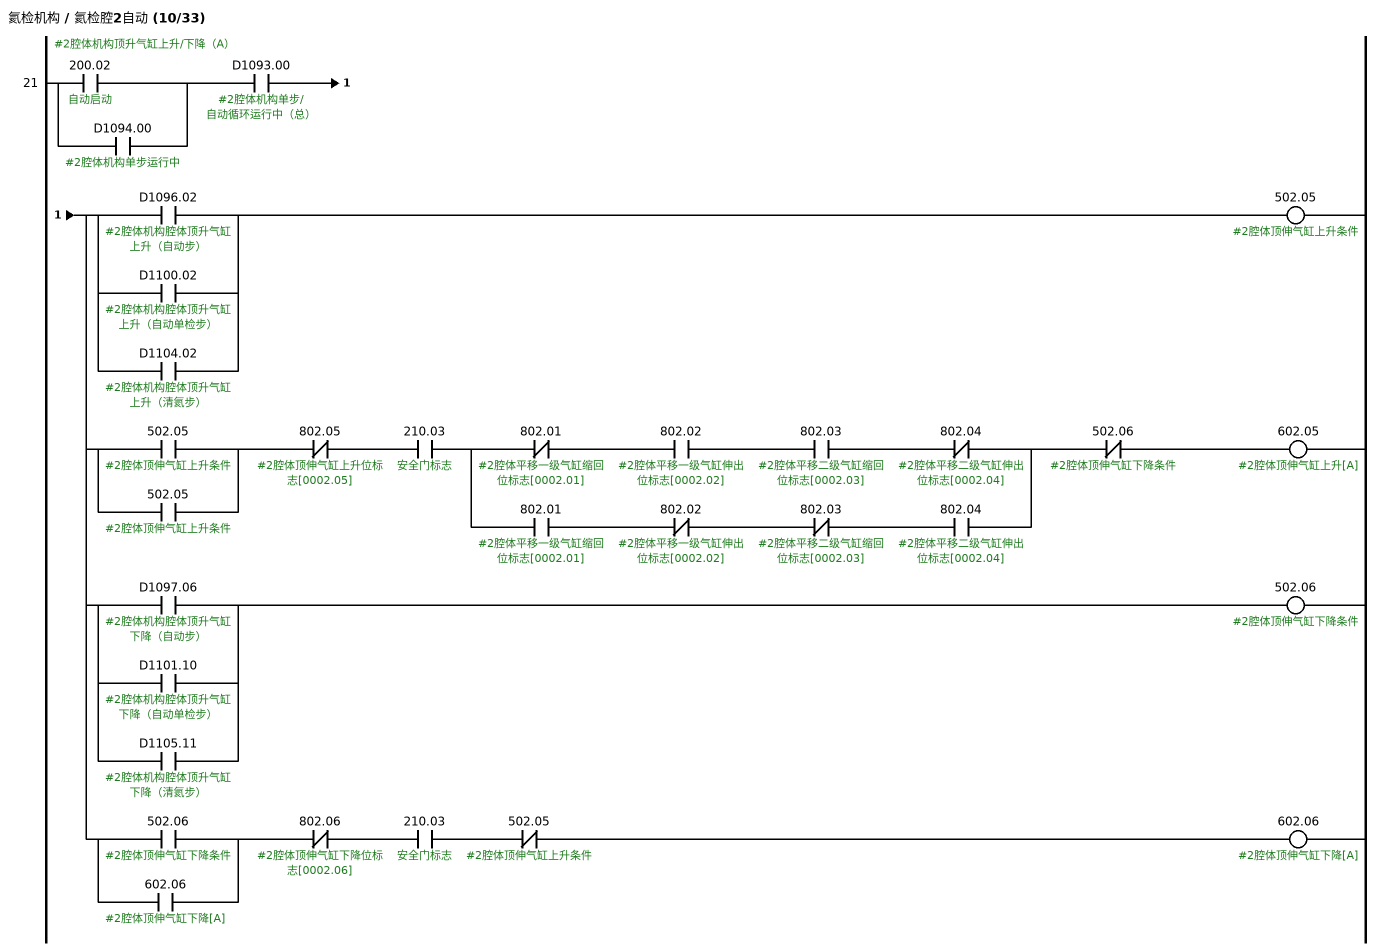
; rung 21: #2腔体机构顶升气缸上升/下降（A）
LD 200.02  ; 自动启动
OR D1094.00  ; #2腔体机构单步运行中
AND D1093.00  ; #2腔体机构单步/自动循环运行中（总）
OUT TR0
LD D1096.02  ; #2腔体机构腔体顶升气缸上升（自动步）
OR D1100.02  ; #2腔体机构腔体顶升气缸上升（自动单检步）
OR D1104.02  ; #2腔体机构腔体顶升气缸上升（清氦步）
ANDLD
OUT 502.05  ; #2腔体顶伸气缸上升条件
LD TR0
LD 502.05  ; #2腔体顶伸气缸上升条件
OR 502.05  ; #2腔体顶伸气缸上升条件
ANDLD
ANDNOT 802.05  ; #2腔体顶伸气缸上升位标志[0002.05]
AND 210.03  ; 安全门标志
LDNOT 802.01  ; #2腔体平移一级气缸缩回位标志[0002.01]
AND 802.02  ; #2腔体平移一级气缸伸出位标志[0002.02]
AND 802.03  ; #2腔体平移二级气缸缩回位标志[0002.03]
ANDNOT 802.04  ; #2腔体平移二级气缸伸出位标志[0002.04]
LD 802.01  ; #2腔体平移一级气缸缩回位标志[0002.01]
ANDNOT 802.02  ; #2腔体平移一级气缸伸出位标志[0002.02]
ANDNOT 802.03  ; #2腔体平移二级气缸缩回位标志[0002.03]
AND 802.04  ; #2腔体平移二级气缸伸出位标志[0002.04]
ORLD
ANDLD
ANDNOT 502.06  ; #2腔体顶伸气缸下降条件
OUT 602.05  ; #2腔体顶伸气缸上升[A]
LD TR0
LD D1097.06  ; #2腔体机构腔体顶升气缸下降（自动步）
OR D1101.10  ; #2腔体机构腔体顶升气缸下降（自动单检步）
OR D1105.11  ; #2腔体机构腔体顶升气缸下降（清氦步）
ANDLD
OUT 502.06  ; #2腔体顶伸气缸下降条件
LD TR0
LD 502.06  ; #2腔体顶伸气缸下降条件
OR 602.06  ; #2腔体顶伸气缸下降[A]
ANDLD
ANDNOT 802.06  ; #2腔体顶伸气缸下降位标志[0002.06]
AND 210.03  ; 安全门标志
ANDNOT 502.05  ; #2腔体顶伸气缸上升条件
OUT 602.06  ; #2腔体顶伸气缸下降[A]

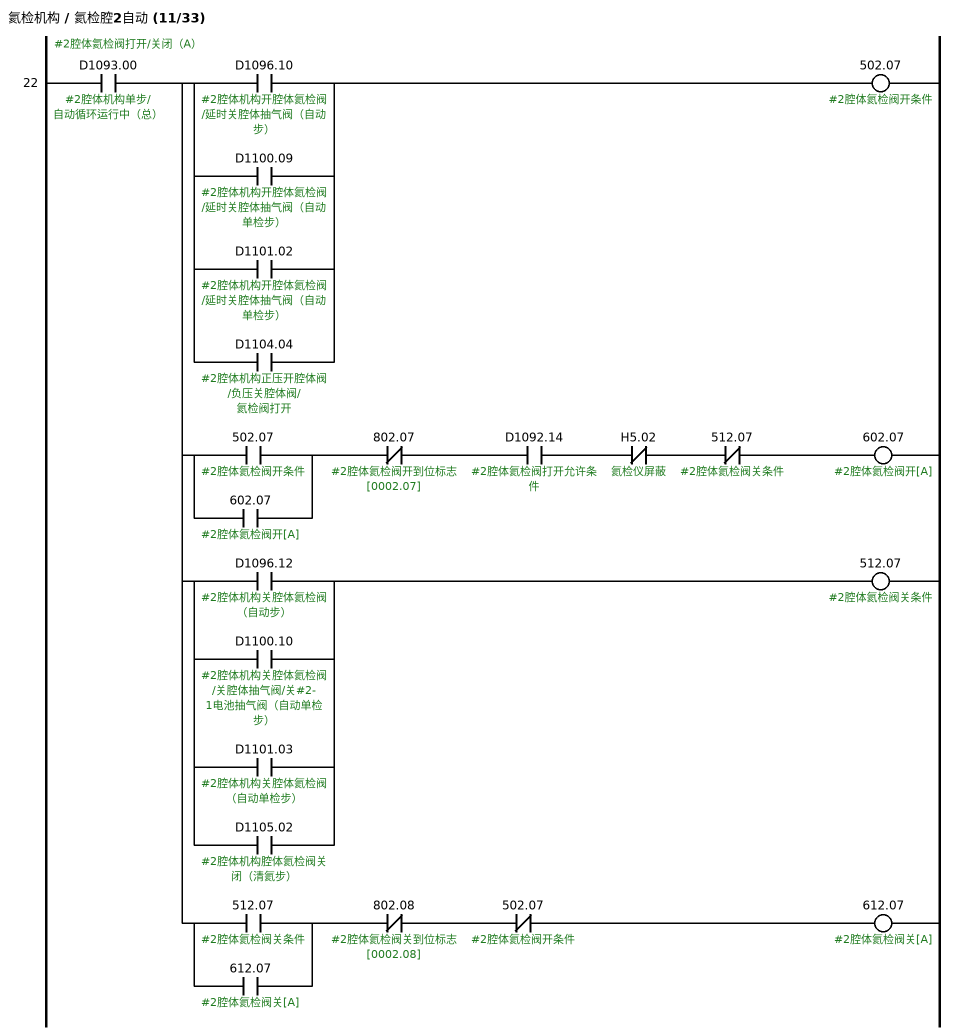
; rung 22: #2腔体氦检阀打开/关闭（A）
LD D1093.00  ; #2腔体机构单步/自动循环运行中（总）
OUT TR0
LD D1096.10  ; #2腔体机构开腔体氦检阀/延时关腔体抽气阀（自动步）
OR D1100.09  ; #2腔体机构开腔体氦检阀/延时关腔体抽气阀（自动单检步）
OR D1101.02  ; #2腔体机构开腔体氦检阀/延时关腔体抽气阀（自动单检步）
OR D1104.04  ; #2腔体机构正压开腔体阀/负压关腔体阀/氦检阀打开
ANDLD
OUT 502.07  ; #2腔体氦检阀开条件
LD TR0
LD 502.07  ; #2腔体氦检阀开条件
OR 602.07  ; #2腔体氦检阀开[A]
ANDLD
ANDNOT 802.07  ; #2腔体氦检阀开到位标志[0002.07]
AND D1092.14  ; #2腔体氦检阀打开允许条件
ANDNOT H5.02  ; 氦检仪屏蔽
ANDNOT 512.07  ; #2腔体氦检阀关条件
OUT 602.07  ; #2腔体氦检阀开[A]
LD TR0
LD D1096.12  ; #2腔体机构关腔体氦检阀（自动步）
OR D1100.10  ; #2腔体机构关腔体氦检阀/关腔体抽气阀/关#2-1电池抽气阀（自动单检步）
OR D1101.03  ; #2腔体机构关腔体氦检阀（自动单检步）
OR D1105.02  ; #2腔体机构腔体氦检阀关闭（清氦步）
ANDLD
OUT 512.07  ; #2腔体氦检阀关条件
LD TR0
LD 512.07  ; #2腔体氦检阀关条件
OR 612.07  ; #2腔体氦检阀关[A]
ANDLD
ANDNOT 802.08  ; #2腔体氦检阀关到位标志[0002.08]
ANDNOT 502.07  ; #2腔体氦检阀开条件
OUT 612.07  ; #2腔体氦检阀关[A]

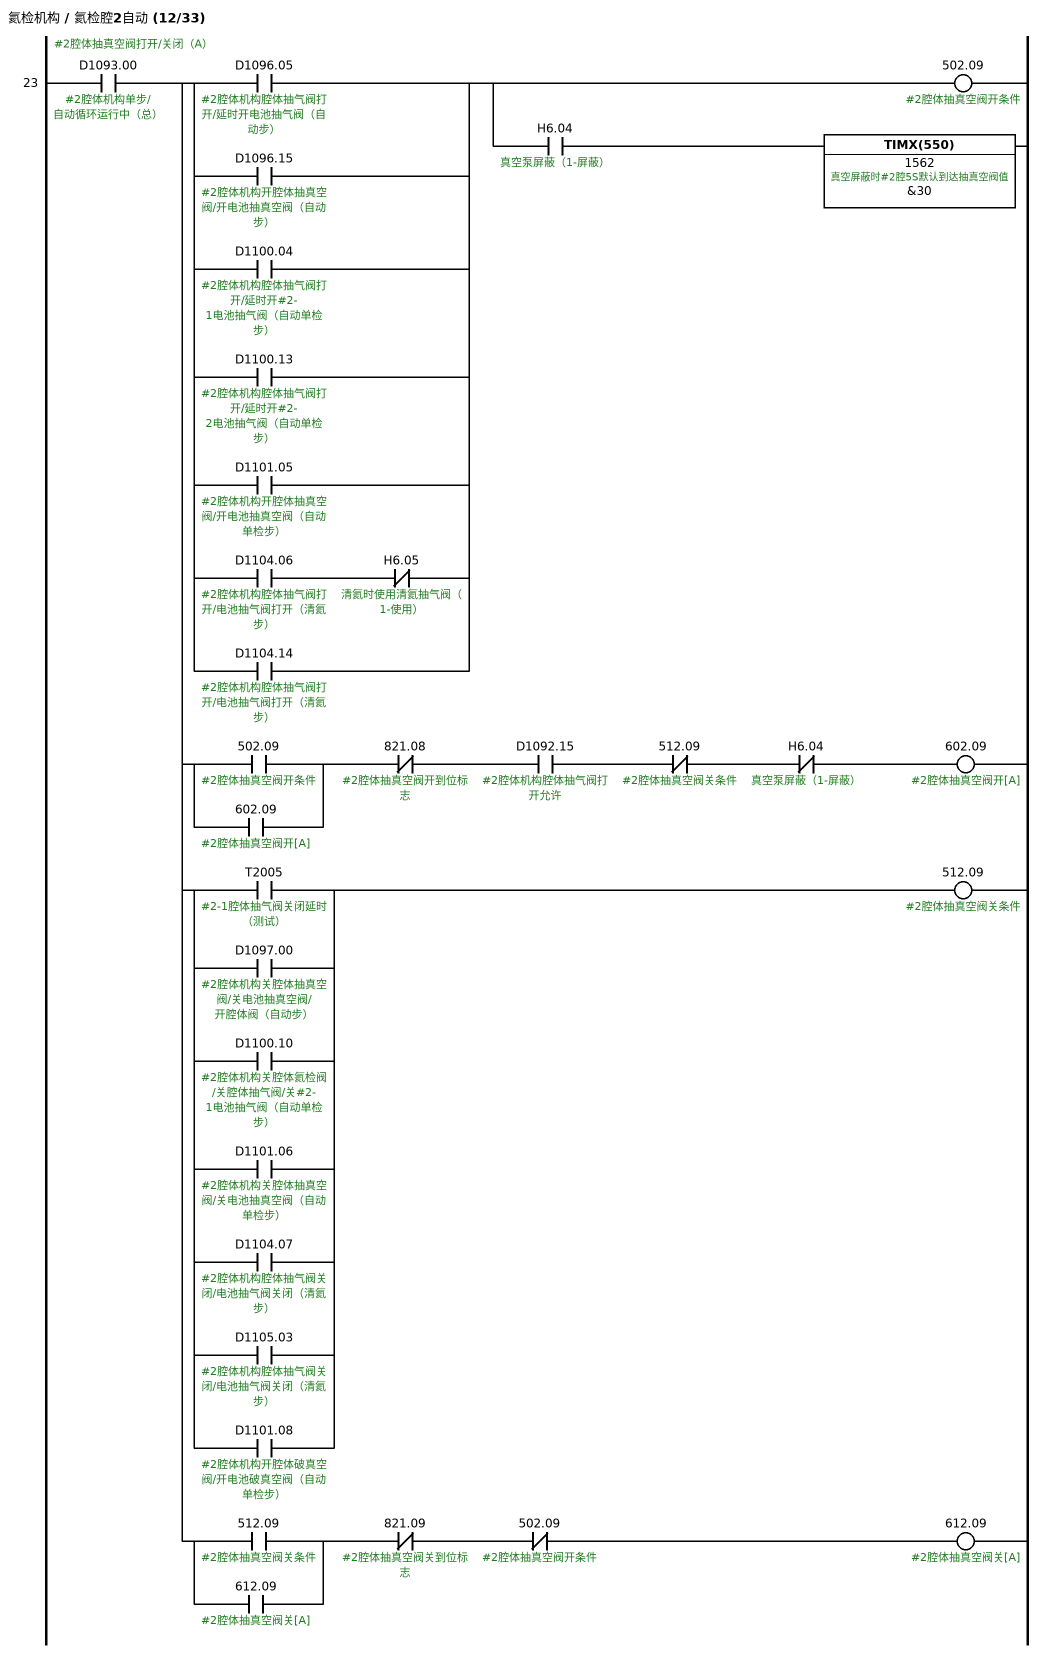
; rung 23: #2腔体抽真空阀打开/关闭（A）
LD D1093.00  ; #2腔体机构单步/自动循环运行中（总）
OUT TR0
LD D1096.05  ; #2腔体机构腔体抽气阀打开/延时开电池抽气阀（自动步）
OR D1096.15  ; #2腔体机构开腔体抽真空阀/开电池抽真空阀（自动步）
OR D1100.04  ; #2腔体机构腔体抽气阀打开/延时开#2-1电池抽气阀（自动单检步）
OR D1100.13  ; #2腔体机构腔体抽气阀打开/延时开#2-2电池抽气阀（自动单检步）
OR D1101.05  ; #2腔体机构开腔体抽真空阀/开电池抽真空阀（自动单检步）
LD D1104.06  ; #2腔体机构腔体抽气阀打开/电池抽气阀打开（清氦步）
ANDNOT H6.05  ; 清氦时使用清氦抽气阀（1-使用）
ORLD
OR D1104.14  ; #2腔体机构腔体抽气阀打开/电池抽气阀打开（清氦步）
ANDLD
OUT 502.09  ; #2腔体抽真空阀开条件
AND H6.04  ; 真空泵屏蔽（1-屏蔽）
TIMX(550) 1562 &30  ; 真空屏蔽时#2腔5S默认到达抽真空阀值
LD TR0
LD 502.09  ; #2腔体抽真空阀开条件
OR 602.09  ; #2腔体抽真空阀开[A]
ANDLD
ANDNOT 821.08  ; #2腔体抽真空阀开到位标志
AND D1092.15  ; #2腔体机构腔体抽气阀打开允许
ANDNOT 512.09  ; #2腔体抽真空阀关条件
ANDNOT H6.04  ; 真空泵屏蔽（1-屏蔽）
OUT 602.09  ; #2腔体抽真空阀开[A]
LD TR0
LD T2005  ; #2-1腔体抽气阀关闭延时（测试）
OR D1097.00  ; #2腔体机构关腔体抽真空阀/关电池抽真空阀/开腔体阀（自动步）
OR D1100.10  ; #2腔体机构关腔体氦检阀/关腔体抽气阀/关#2-1电池抽气阀（自动单检步）
OR D1101.06  ; #2腔体机构关腔体抽真空阀/关电池抽真空阀（自动单检步）
OR D1104.07  ; #2腔体机构腔体抽气阀关闭/电池抽气阀关闭（清氦步）
OR D1105.03  ; #2腔体机构腔体抽气阀关闭/电池抽气阀关闭（清氦步）
OR D1101.08  ; #2腔体机构开腔体破真空阀/开电池破真空阀（自动单检步）
ANDLD
OUT 512.09  ; #2腔体抽真空阀关条件
LD TR0
LD 512.09  ; #2腔体抽真空阀关条件
OR 612.09  ; #2腔体抽真空阀关[A]
ANDLD
ANDNOT 821.09  ; #2腔体抽真空阀关到位标志
ANDNOT 502.09  ; #2腔体抽真空阀开条件
OUT 612.09  ; #2腔体抽真空阀关[A]

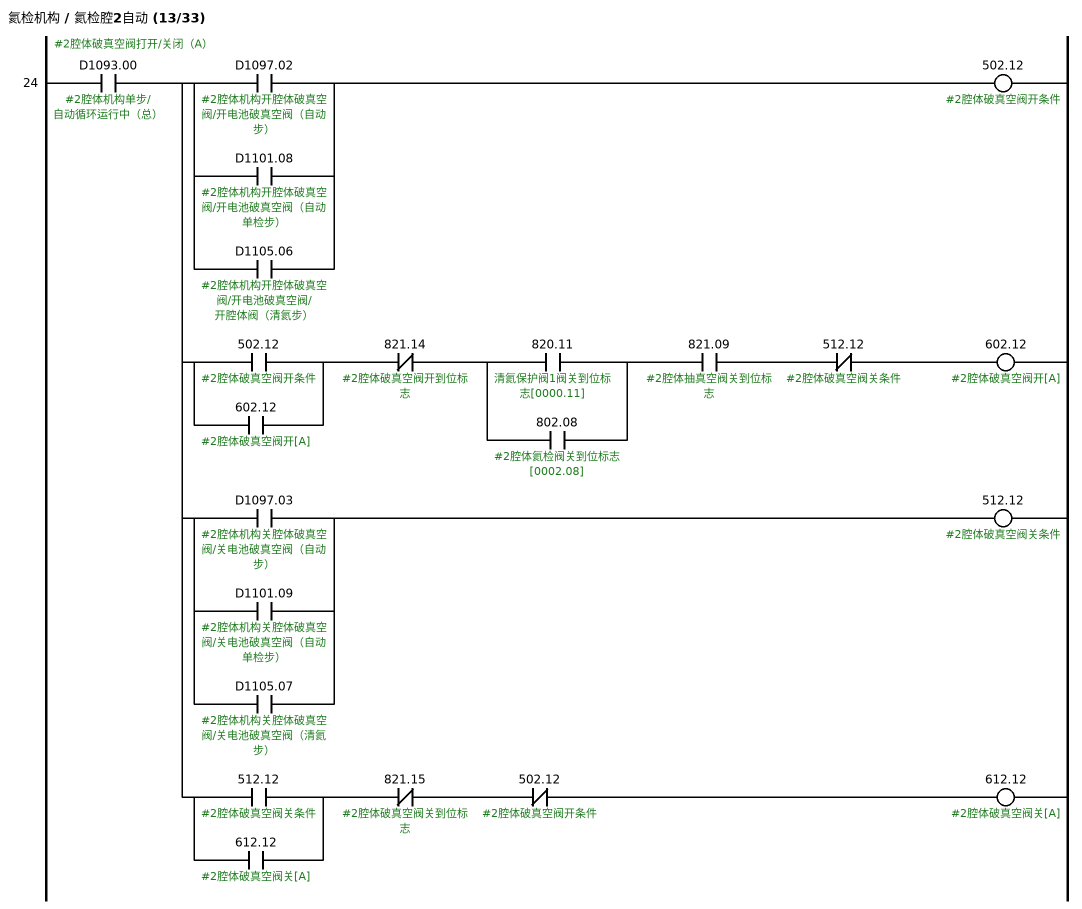
; rung 24: #2腔体破真空阀打开/关闭（A）
LD D1093.00  ; #2腔体机构单步/自动循环运行中（总）
OUT TR0
LD D1097.02  ; #2腔体机构开腔体破真空阀/开电池破真空阀（自动步）
OR D1101.08  ; #2腔体机构开腔体破真空阀/开电池破真空阀（自动单检步）
OR D1105.06  ; #2腔体机构开腔体破真空阀/开电池破真空阀/开腔体阀（清氦步）
ANDLD
OUT 502.12  ; #2腔体破真空阀开条件
LD TR0
LD 502.12  ; #2腔体破真空阀开条件
OR 602.12  ; #2腔体破真空阀开[A]
ANDLD
ANDNOT 821.14  ; #2腔体破真空阀开到位标志
LD 820.11  ; 清氦保护阀1阀关到位标志[0000.11]
OR 802.08  ; #2腔体氦检阀关到位标志[0002.08]
ANDLD
AND 821.09  ; #2腔体抽真空阀关到位标志
ANDNOT 512.12  ; #2腔体破真空阀关条件
OUT 602.12  ; #2腔体破真空阀开[A]
LD TR0
LD D1097.03  ; #2腔体机构关腔体破真空阀/关电池破真空阀（自动步）
OR D1101.09  ; #2腔体机构关腔体破真空阀/关电池破真空阀（自动单检步）
OR D1105.07  ; #2腔体机构关腔体破真空阀/关电池破真空阀（清氦步）
ANDLD
OUT 512.12  ; #2腔体破真空阀关条件
LD TR0
LD 512.12  ; #2腔体破真空阀关条件
OR 612.12  ; #2腔体破真空阀关[A]
ANDLD
ANDNOT 821.15  ; #2腔体破真空阀关到位标志
ANDNOT 502.12  ; #2腔体破真空阀开条件
OUT 612.12  ; #2腔体破真空阀关[A]

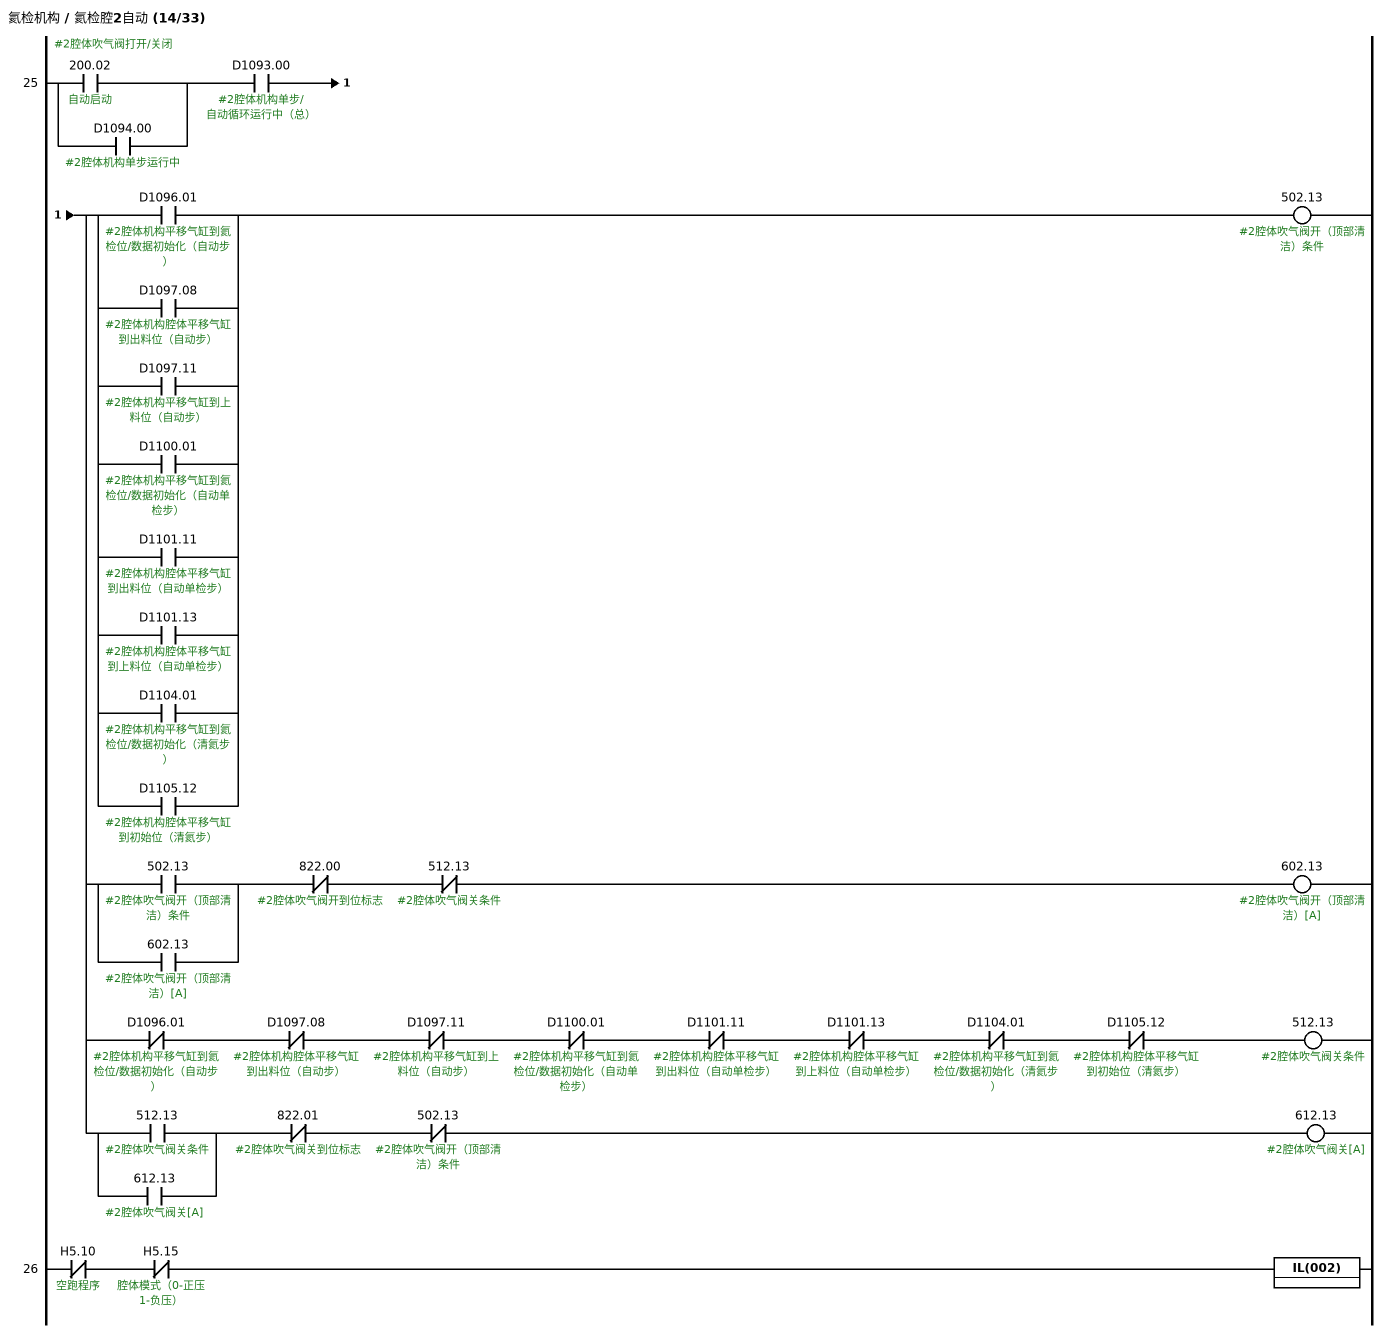
; rung 25: #2腔体吹气阀打开/关闭
LD 200.02  ; 自动启动
OR D1094.00  ; #2腔体机构单步运行中
AND D1093.00  ; #2腔体机构单步/自动循环运行中（总）
OUT TR0
LD D1096.01  ; #2腔体机构平移气缸到氦检位/数据初始化（自动步）
OR D1097.08  ; #2腔体机构腔体平移气缸到出料位（自动步）
OR D1097.11  ; #2腔体机构平移气缸到上料位（自动步）
OR D1100.01  ; #2腔体机构平移气缸到氦检位/数据初始化（自动单检步）
OR D1101.11  ; #2腔体机构腔体平移气缸到出料位（自动单检步）
OR D1101.13  ; #2腔体机构腔体平移气缸到上料位（自动单检步）
OR D1104.01  ; #2腔体机构平移气缸到氦检位/数据初始化（清氦步）
OR D1105.12  ; #2腔体机构腔体平移气缸到初始位（清氦步）
ANDLD
OUT 502.13  ; #2腔体吹气阀开（顶部清洁）条件
LD TR0
LD 502.13  ; #2腔体吹气阀开（顶部清洁）条件
OR 602.13  ; #2腔体吹气阀开（顶部清洁）[A]
ANDLD
ANDNOT 822.00  ; #2腔体吹气阀开到位标志
ANDNOT 512.13  ; #2腔体吹气阀关条件
OUT 602.13  ; #2腔体吹气阀开（顶部清洁）[A]
LD TR0
ANDNOT D1096.01  ; #2腔体机构平移气缸到氦检位/数据初始化（自动步）
ANDNOT D1097.08  ; #2腔体机构腔体平移气缸到出料位（自动步）
ANDNOT D1097.11  ; #2腔体机构平移气缸到上料位（自动步）
ANDNOT D1100.01  ; #2腔体机构平移气缸到氦检位/数据初始化（自动单检步）
ANDNOT D1101.11  ; #2腔体机构腔体平移气缸到出料位（自动单检步）
ANDNOT D1101.13  ; #2腔体机构腔体平移气缸到上料位（自动单检步）
ANDNOT D1104.01  ; #2腔体机构平移气缸到氦检位/数据初始化（清氦步）
ANDNOT D1105.12  ; #2腔体机构腔体平移气缸到初始位（清氦步）
OUT 512.13  ; #2腔体吹气阀关条件
LD TR0
LD 512.13  ; #2腔体吹气阀关条件
OR 612.13  ; #2腔体吹气阀关[A]
ANDLD
ANDNOT 822.01  ; #2腔体吹气阀关到位标志
ANDNOT 502.13  ; #2腔体吹气阀开（顶部清洁）条件
OUT 612.13  ; #2腔体吹气阀关[A]
; rung 26
LDNOT H5.10  ; 空跑程序
ANDNOT H5.15  ; 腔体模式（0-正压 1-负压）
IL(002)

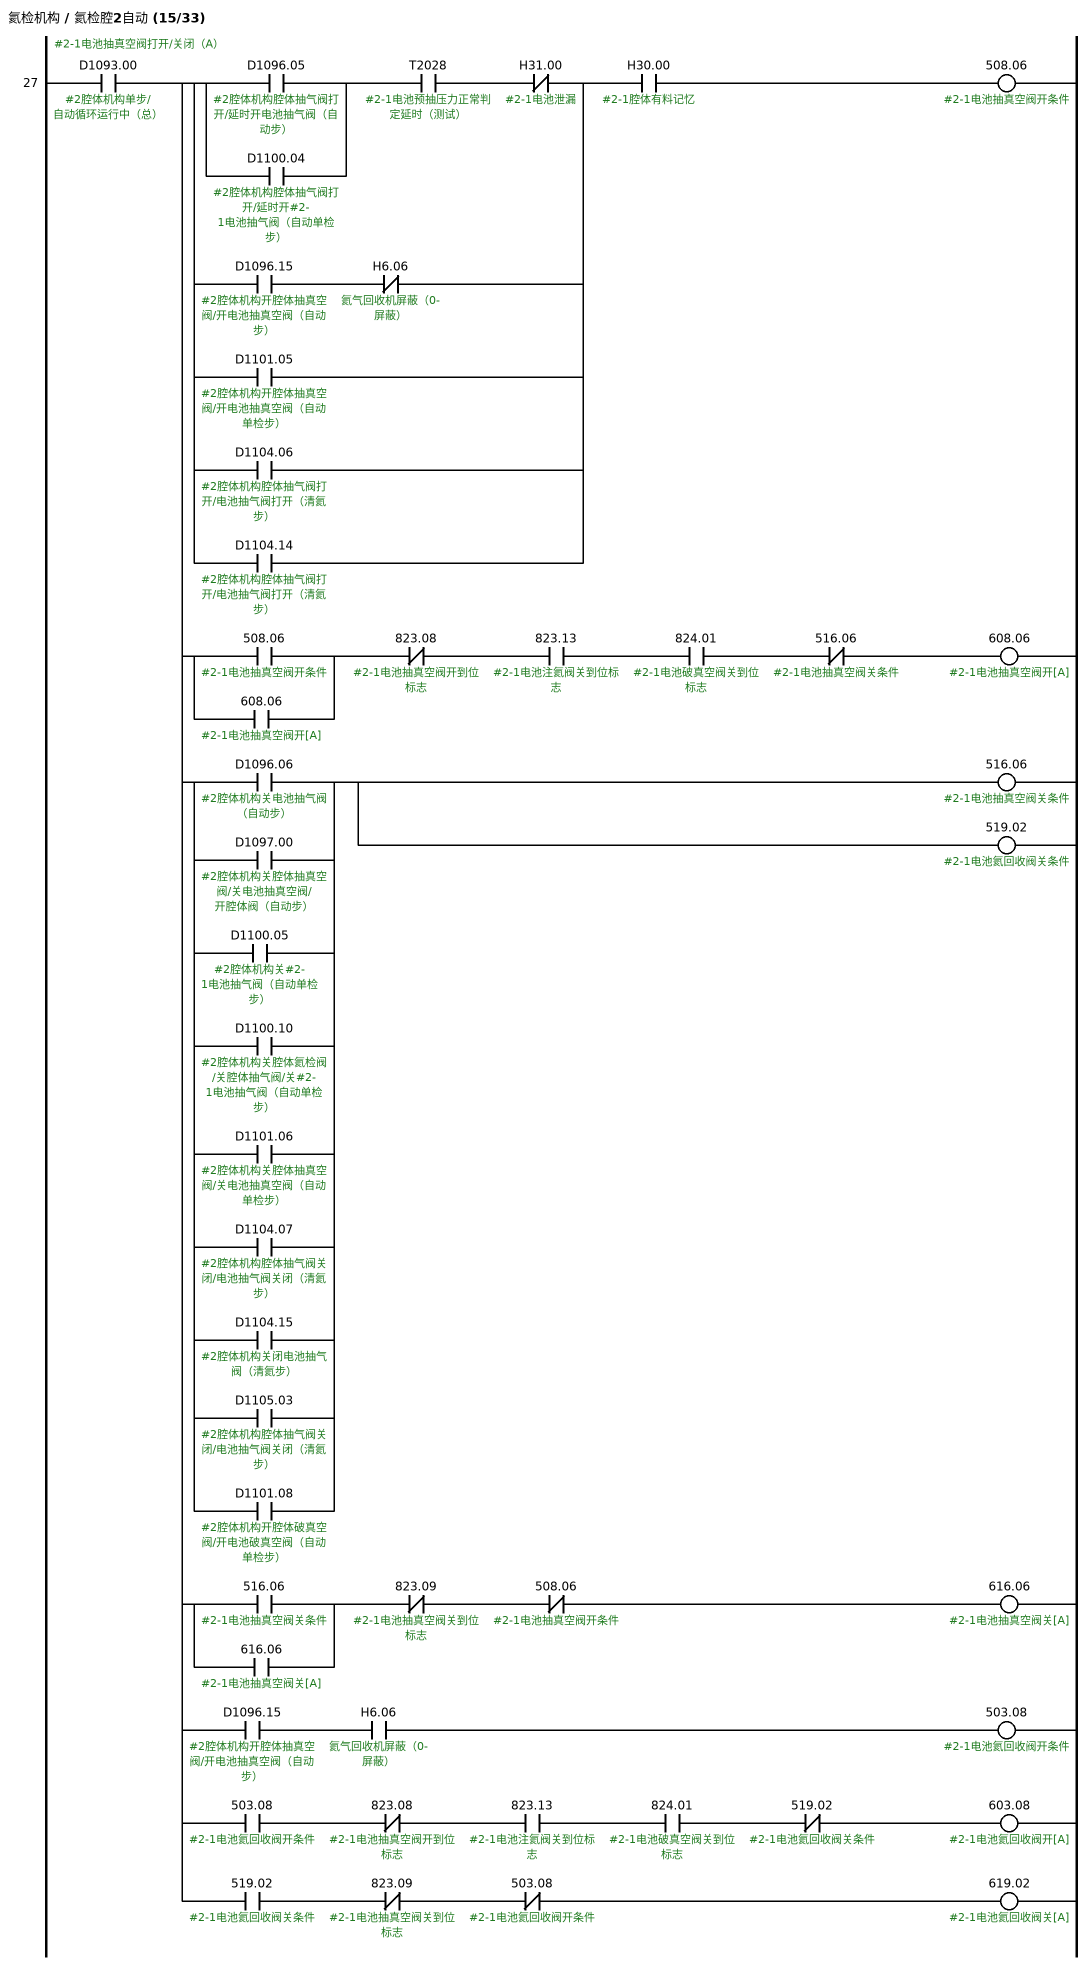
; rung 27: #2-1电池抽真空阀打开/关闭（A）
LD D1093.00  ; #2腔体机构单步/自动循环运行中（总）
OUT TR0
LD D1096.05  ; #2腔体机构腔体抽气阀打开/延时开电池抽气阀（自动步）
OR D1100.04  ; #2腔体机构腔体抽气阀打开/延时开#2-1电池抽气阀（自动单检步）
AND T2028  ; #2-1电池预抽压力正常判定延时（测试）
ANDNOT H31.00  ; #2-1电池泄漏
LD D1096.15  ; #2腔体机构开腔体抽真空阀/开电池抽真空阀（自动步）
ANDNOT H6.06  ; 氦气回收机屏蔽（0-屏蔽）
ORLD
OR D1101.05  ; #2腔体机构开腔体抽真空阀/开电池抽真空阀（自动单检步）
OR D1104.06  ; #2腔体机构腔体抽气阀打开/电池抽气阀打开（清氦步）
OR D1104.14  ; #2腔体机构腔体抽气阀打开/电池抽气阀打开（清氦步）
ANDLD
AND H30.00  ; #2-1腔体有料记忆
OUT 508.06  ; #2-1电池抽真空阀开条件
LD TR0
LD 508.06  ; #2-1电池抽真空阀开条件
OR 608.06  ; #2-1电池抽真空阀开[A]
ANDLD
ANDNOT 823.08  ; #2-1电池抽真空阀开到位标志
AND 823.13  ; #2-1电池注氦阀关到位标志
AND 824.01  ; #2-1电池破真空阀关到位标志
ANDNOT 516.06  ; #2-1电池抽真空阀关条件
OUT 608.06  ; #2-1电池抽真空阀开[A]
LD TR0
LD D1096.06  ; #2腔体机构关电池抽气阀（自动步）
OR D1097.00  ; #2腔体机构关腔体抽真空阀/关电池抽真空阀/开腔体阀（自动步）
OR D1100.05  ; #2腔体机构关#2-1电池抽气阀（自动单检步）
OR D1100.10  ; #2腔体机构关腔体氦检阀/关腔体抽气阀/关#2-1电池抽气阀（自动单检步）
OR D1101.06  ; #2腔体机构关腔体抽真空阀/关电池抽真空阀（自动单检步）
OR D1104.07  ; #2腔体机构腔体抽气阀关闭/电池抽气阀关闭（清氦步）
OR D1104.15  ; #2腔体机构关闭电池抽气阀（清氦步）
OR D1105.03  ; #2腔体机构腔体抽气阀关闭/电池抽气阀关闭（清氦步）
OR D1101.08  ; #2腔体机构开腔体破真空阀/开电池破真空阀（自动单检步）
ANDLD
OUT 516.06  ; #2-1电池抽真空阀关条件
OUT 519.02  ; #2-1电池氦回收阀关条件
LD TR0
LD 516.06  ; #2-1电池抽真空阀关条件
OR 616.06  ; #2-1电池抽真空阀关[A]
ANDLD
ANDNOT 823.09  ; #2-1电池抽真空阀关到位标志
ANDNOT 508.06  ; #2-1电池抽真空阀开条件
OUT 616.06  ; #2-1电池抽真空阀关[A]
LD TR0
AND D1096.15  ; #2腔体机构开腔体抽真空阀/开电池抽真空阀（自动步）
AND H6.06  ; 氦气回收机屏蔽（0-屏蔽）
OUT 503.08  ; #2-1电池氦回收阀开条件
LD TR0
AND 503.08  ; #2-1电池氦回收阀开条件
ANDNOT 823.08  ; #2-1电池抽真空阀开到位标志
AND 823.13  ; #2-1电池注氦阀关到位标志
AND 824.01  ; #2-1电池破真空阀关到位标志
ANDNOT 519.02  ; #2-1电池氦回收阀关条件
OUT 603.08  ; #2-1电池氦回收阀开[A]
LD TR0
AND 519.02  ; #2-1电池氦回收阀关条件
ANDNOT 823.09  ; #2-1电池抽真空阀关到位标志
ANDNOT 503.08  ; #2-1电池氦回收阀开条件
OUT 619.02  ; #2-1电池氦回收阀关[A]

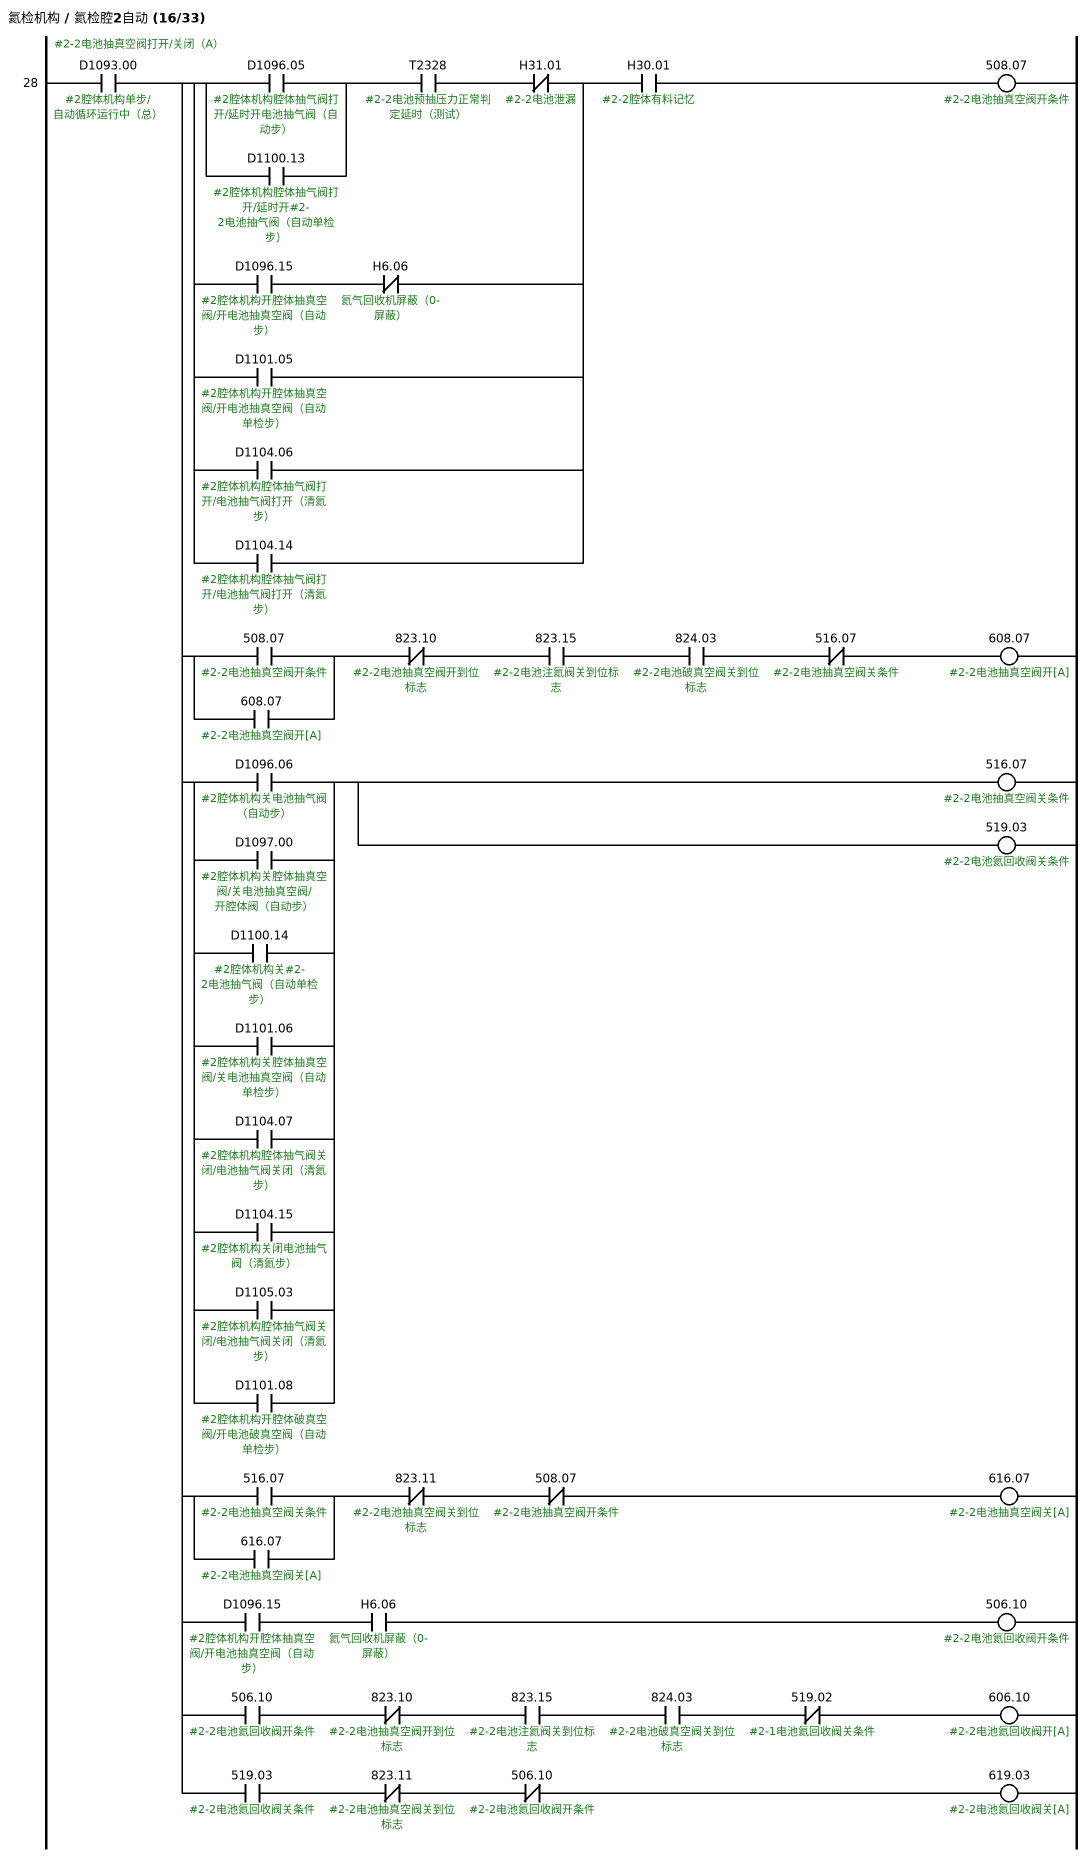
; rung 28: #2-2电池抽真空阀打开/关闭（A）
LD D1093.00  ; #2腔体机构单步/自动循环运行中（总）
OUT TR0
LD D1096.05  ; #2腔体机构腔体抽气阀打开/延时开电池抽气阀（自动步）
OR D1100.13  ; #2腔体机构腔体抽气阀打开/延时开#2-2电池抽气阀（自动单检步）
AND T2328  ; #2-2电池预抽压力正常判定延时（测试）
ANDNOT H31.01  ; #2-2电池泄漏
LD D1096.15  ; #2腔体机构开腔体抽真空阀/开电池抽真空阀（自动步）
ANDNOT H6.06  ; 氦气回收机屏蔽（0-屏蔽）
ORLD
OR D1101.05  ; #2腔体机构开腔体抽真空阀/开电池抽真空阀（自动单检步）
OR D1104.06  ; #2腔体机构腔体抽气阀打开/电池抽气阀打开（清氦步）
OR D1104.14  ; #2腔体机构腔体抽气阀打开/电池抽气阀打开（清氦步）
ANDLD
AND H30.01  ; #2-2腔体有料记忆
OUT 508.07  ; #2-2电池抽真空阀开条件
LD TR0
LD 508.07  ; #2-2电池抽真空阀开条件
OR 608.07  ; #2-2电池抽真空阀开[A]
ANDLD
ANDNOT 823.10  ; #2-2电池抽真空阀开到位标志
AND 823.15  ; #2-2电池注氦阀关到位标志
AND 824.03  ; #2-2电池破真空阀关到位标志
ANDNOT 516.07  ; #2-2电池抽真空阀关条件
OUT 608.07  ; #2-2电池抽真空阀开[A]
LD TR0
LD D1096.06  ; #2腔体机构关电池抽气阀（自动步）
OR D1097.00  ; #2腔体机构关腔体抽真空阀/关电池抽真空阀/开腔体阀（自动步）
OR D1100.14  ; #2腔体机构关#2-2电池抽气阀（自动单检步）
OR D1101.06  ; #2腔体机构关腔体抽真空阀/关电池抽真空阀（自动单检步）
OR D1104.07  ; #2腔体机构腔体抽气阀关闭/电池抽气阀关闭（清氦步）
OR D1104.15  ; #2腔体机构关闭电池抽气阀（清氦步）
OR D1105.03  ; #2腔体机构腔体抽气阀关闭/电池抽气阀关闭（清氦步）
OR D1101.08  ; #2腔体机构开腔体破真空阀/开电池破真空阀（自动单检步）
ANDLD
OUT 516.07  ; #2-2电池抽真空阀关条件
OUT 519.03  ; #2-2电池氦回收阀关条件
LD TR0
LD 516.07  ; #2-2电池抽真空阀关条件
OR 616.07  ; #2-2电池抽真空阀关[A]
ANDLD
ANDNOT 823.11  ; #2-2电池抽真空阀关到位标志
ANDNOT 508.07  ; #2-2电池抽真空阀开条件
OUT 616.07  ; #2-2电池抽真空阀关[A]
LD TR0
AND D1096.15  ; #2腔体机构开腔体抽真空阀/开电池抽真空阀（自动步）
AND H6.06  ; 氦气回收机屏蔽（0-屏蔽）
OUT 506.10  ; #2-2电池氦回收阀开条件
LD TR0
AND 506.10  ; #2-2电池氦回收阀开条件
ANDNOT 823.10  ; #2-2电池抽真空阀开到位标志
AND 823.15  ; #2-2电池注氦阀关到位标志
AND 824.03  ; #2-2电池破真空阀关到位标志
ANDNOT 519.02  ; #2-1电池氦回收阀关条件
OUT 606.10  ; #2-2电池氦回收阀开[A]
LD TR0
AND 519.03  ; #2-2电池氦回收阀关条件
ANDNOT 823.11  ; #2-2电池抽真空阀关到位标志
ANDNOT 506.10  ; #2-2电池氦回收阀开条件
OUT 619.03  ; #2-2电池氦回收阀关[A]

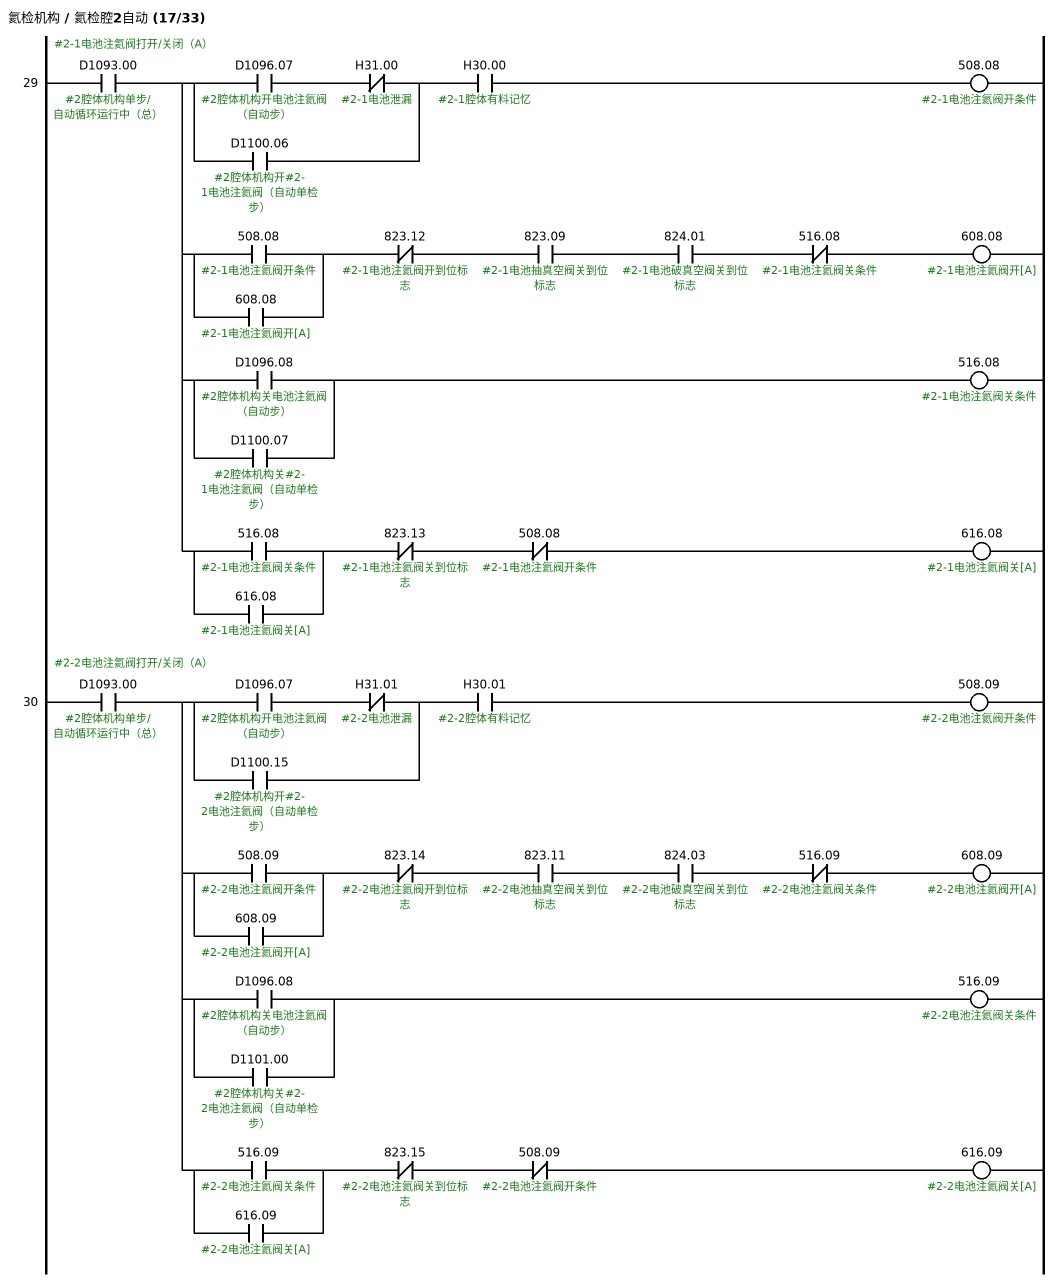
; rung 29: #2-1电池注氦阀打开/关闭（A）
LD D1093.00  ; #2腔体机构单步/自动循环运行中（总）
OUT TR0
LD D1096.07  ; #2腔体机构开电池注氦阀（自动步）
ANDNOT H31.00  ; #2-1电池泄漏
OR D1100.06  ; #2腔体机构开#2-1电池注氦阀（自动单检步）
ANDLD
AND H30.00  ; #2-1腔体有料记忆
OUT 508.08  ; #2-1电池注氦阀开条件
LD TR0
LD 508.08  ; #2-1电池注氦阀开条件
OR 608.08  ; #2-1电池注氦阀开[A]
ANDLD
ANDNOT 823.12  ; #2-1电池注氦阀开到位标志
AND 823.09  ; #2-1电池抽真空阀关到位标志
AND 824.01  ; #2-1电池破真空阀关到位标志
ANDNOT 516.08  ; #2-1电池注氦阀关条件
OUT 608.08  ; #2-1电池注氦阀开[A]
LD TR0
LD D1096.08  ; #2腔体机构关电池注氦阀（自动步）
OR D1100.07  ; #2腔体机构关#2-1电池注氦阀（自动单检步）
ANDLD
OUT 516.08  ; #2-1电池注氦阀关条件
LD TR0
LD 516.08  ; #2-1电池注氦阀关条件
OR 616.08  ; #2-1电池注氦阀关[A]
ANDLD
ANDNOT 823.13  ; #2-1电池注氦阀关到位标志
ANDNOT 508.08  ; #2-1电池注氦阀开条件
OUT 616.08  ; #2-1电池注氦阀关[A]
; rung 30: #2-2电池注氦阀打开/关闭（A）
LD D1093.00  ; #2腔体机构单步/自动循环运行中（总）
OUT TR0
LD D1096.07  ; #2腔体机构开电池注氦阀（自动步）
ANDNOT H31.01  ; #2-2电池泄漏
OR D1100.15  ; #2腔体机构开#2-2电池注氦阀（自动单检步）
ANDLD
AND H30.01  ; #2-2腔体有料记忆
OUT 508.09  ; #2-2电池注氦阀开条件
LD TR0
LD 508.09  ; #2-2电池注氦阀开条件
OR 608.09  ; #2-2电池注氦阀开[A]
ANDLD
ANDNOT 823.14  ; #2-2电池注氦阀开到位标志
AND 823.11  ; #2-2电池抽真空阀关到位标志
AND 824.03  ; #2-2电池破真空阀关到位标志
ANDNOT 516.09  ; #2-2电池注氦阀关条件
OUT 608.09  ; #2-2电池注氦阀开[A]
LD TR0
LD D1096.08  ; #2腔体机构关电池注氦阀（自动步）
OR D1101.00  ; #2腔体机构关#2-2电池注氦阀（自动单检步）
ANDLD
OUT 516.09  ; #2-2电池注氦阀关条件
LD TR0
LD 516.09  ; #2-2电池注氦阀关条件
OR 616.09  ; #2-2电池注氦阀关[A]
ANDLD
ANDNOT 823.15  ; #2-2电池注氦阀关到位标志
ANDNOT 508.09  ; #2-2电池注氦阀开条件
OUT 616.09  ; #2-2电池注氦阀关[A]

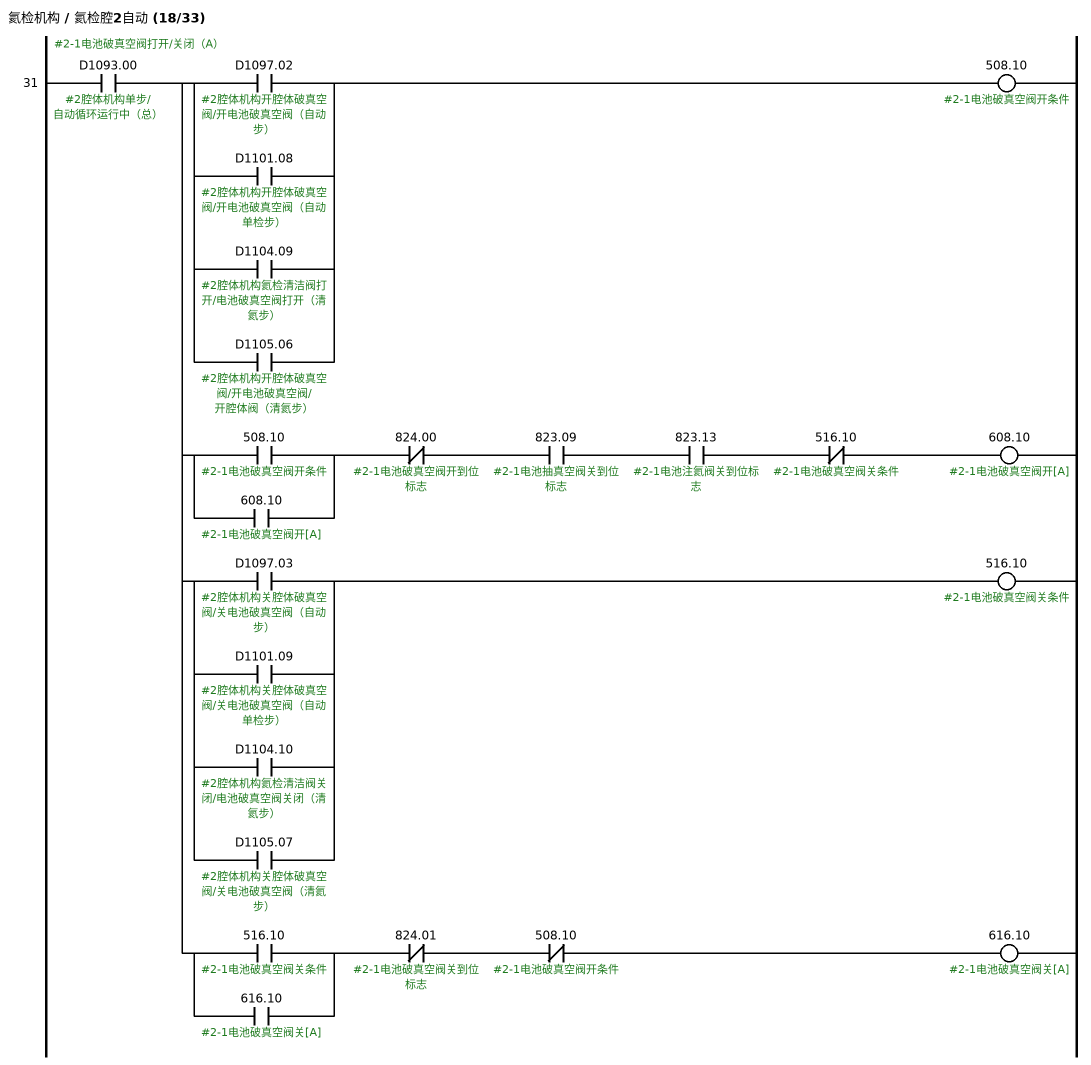
; rung 31: #2-1电池破真空阀打开/关闭（A）
LD D1093.00  ; #2腔体机构单步/自动循环运行中（总）
OUT TR0
LD D1097.02  ; #2腔体机构开腔体破真空阀/开电池破真空阀（自动步）
OR D1101.08  ; #2腔体机构开腔体破真空阀/开电池破真空阀（自动单检步）
OR D1104.09  ; #2腔体机构氦检清洁阀打开/电池破真空阀打开（清氦步）
OR D1105.06  ; #2腔体机构开腔体破真空阀/开电池破真空阀/开腔体阀（清氦步）
ANDLD
OUT 508.10  ; #2-1电池破真空阀开条件
LD TR0
LD 508.10  ; #2-1电池破真空阀开条件
OR 608.10  ; #2-1电池破真空阀开[A]
ANDLD
ANDNOT 824.00  ; #2-1电池破真空阀开到位标志
AND 823.09  ; #2-1电池抽真空阀关到位标志
AND 823.13  ; #2-1电池注氦阀关到位标志
ANDNOT 516.10  ; #2-1电池破真空阀关条件
OUT 608.10  ; #2-1电池破真空阀开[A]
LD TR0
LD D1097.03  ; #2腔体机构关腔体破真空阀/关电池破真空阀（自动步）
OR D1101.09  ; #2腔体机构关腔体破真空阀/关电池破真空阀（自动单检步）
OR D1104.10  ; #2腔体机构氦检清洁阀关闭/电池破真空阀关闭（清氦步）
OR D1105.07  ; #2腔体机构关腔体破真空阀/关电池破真空阀（清氦步）
ANDLD
OUT 516.10  ; #2-1电池破真空阀关条件
LD TR0
LD 516.10  ; #2-1电池破真空阀关条件
OR 616.10  ; #2-1电池破真空阀关[A]
ANDLD
ANDNOT 824.01  ; #2-1电池破真空阀关到位标志
ANDNOT 508.10  ; #2-1电池破真空阀开条件
OUT 616.10  ; #2-1电池破真空阀关[A]

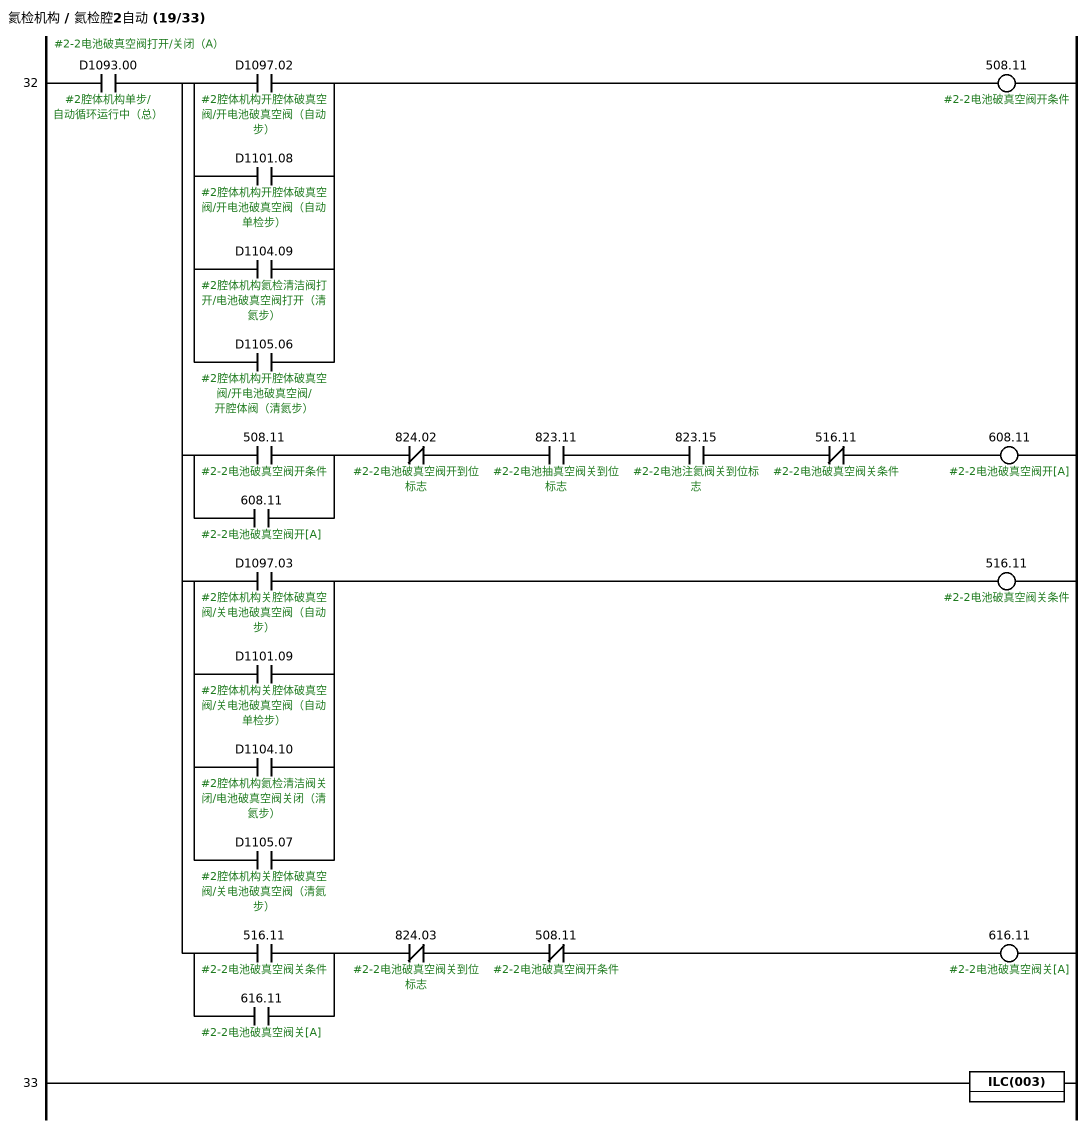
; rung 32: #2-2电池破真空阀打开/关闭（A）
LD D1093.00  ; #2腔体机构单步/自动循环运行中（总）
OUT TR0
LD D1097.02  ; #2腔体机构开腔体破真空阀/开电池破真空阀（自动步）
OR D1101.08  ; #2腔体机构开腔体破真空阀/开电池破真空阀（自动单检步）
OR D1104.09  ; #2腔体机构氦检清洁阀打开/电池破真空阀打开（清氦步）
OR D1105.06  ; #2腔体机构开腔体破真空阀/开电池破真空阀/开腔体阀（清氦步）
ANDLD
OUT 508.11  ; #2-2电池破真空阀开条件
LD TR0
LD 508.11  ; #2-2电池破真空阀开条件
OR 608.11  ; #2-2电池破真空阀开[A]
ANDLD
ANDNOT 824.02  ; #2-2电池破真空阀开到位标志
AND 823.11  ; #2-2电池抽真空阀关到位标志
AND 823.15  ; #2-2电池注氦阀关到位标志
ANDNOT 516.11  ; #2-2电池破真空阀关条件
OUT 608.11  ; #2-2电池破真空阀开[A]
LD TR0
LD D1097.03  ; #2腔体机构关腔体破真空阀/关电池破真空阀（自动步）
OR D1101.09  ; #2腔体机构关腔体破真空阀/关电池破真空阀（自动单检步）
OR D1104.10  ; #2腔体机构氦检清洁阀关闭/电池破真空阀关闭（清氦步）
OR D1105.07  ; #2腔体机构关腔体破真空阀/关电池破真空阀（清氦步）
ANDLD
OUT 516.11  ; #2-2电池破真空阀关条件
LD TR0
LD 516.11  ; #2-2电池破真空阀关条件
OR 616.11  ; #2-2电池破真空阀关[A]
ANDLD
ANDNOT 824.03  ; #2-2电池破真空阀关到位标志
ANDNOT 508.11  ; #2-2电池破真空阀开条件
OUT 616.11  ; #2-2电池破真空阀关[A]
; rung 33
ILC(003)

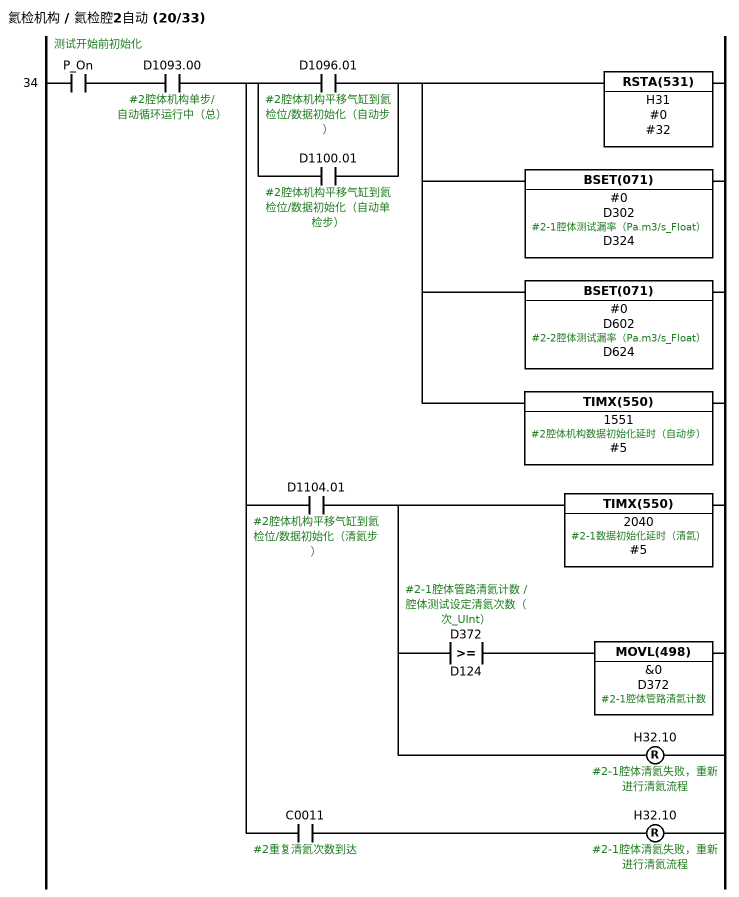
; rung 34: 测试开始前初始化
LD P_On
AND D1093.00  ; #2腔体机构单步/自动循环运行中（总）
OUT TR0
LD D1096.01  ; #2腔体机构平移气缸到氦检位/数据初始化（自动步）
OR D1100.01  ; #2腔体机构平移气缸到氦检位/数据初始化（自动单检步）
ANDLD
RSTA(531) H31 #0 #32
BSET(071) #0 D302 D324  ; #2-1腔体测试漏率（Pa.m3/s_Float）
BSET(071) #0 D602 D624  ; #2-2腔体测试漏率（Pa.m3/s_Float）
TIMX(550) 1551 #5  ; #2腔体机构数据初始化延时（自动步）
LD TR0
AND D1104.01  ; #2腔体机构平移气缸到氦检位/数据初始化（清氦步）
OUT TR1
TIMX(550) 2040 #5  ; #2-1数据初始化延时（清氦）
AND>=(325) D372 D124  ; #2-1腔体管路清氦计数, 腔体测试设定清氦次数（次_UInt）
MOVL(498) &0 D372  ; #2-1腔体管路清氦计数
LD TR1
RSET H32.10  ; #2-1腔体清氦失败，重新进行清氦流程
LD TR0
AND C0011  ; #2重复清氦次数到达
RSET H32.10  ; #2-1腔体清氦失败，重新进行清氦流程

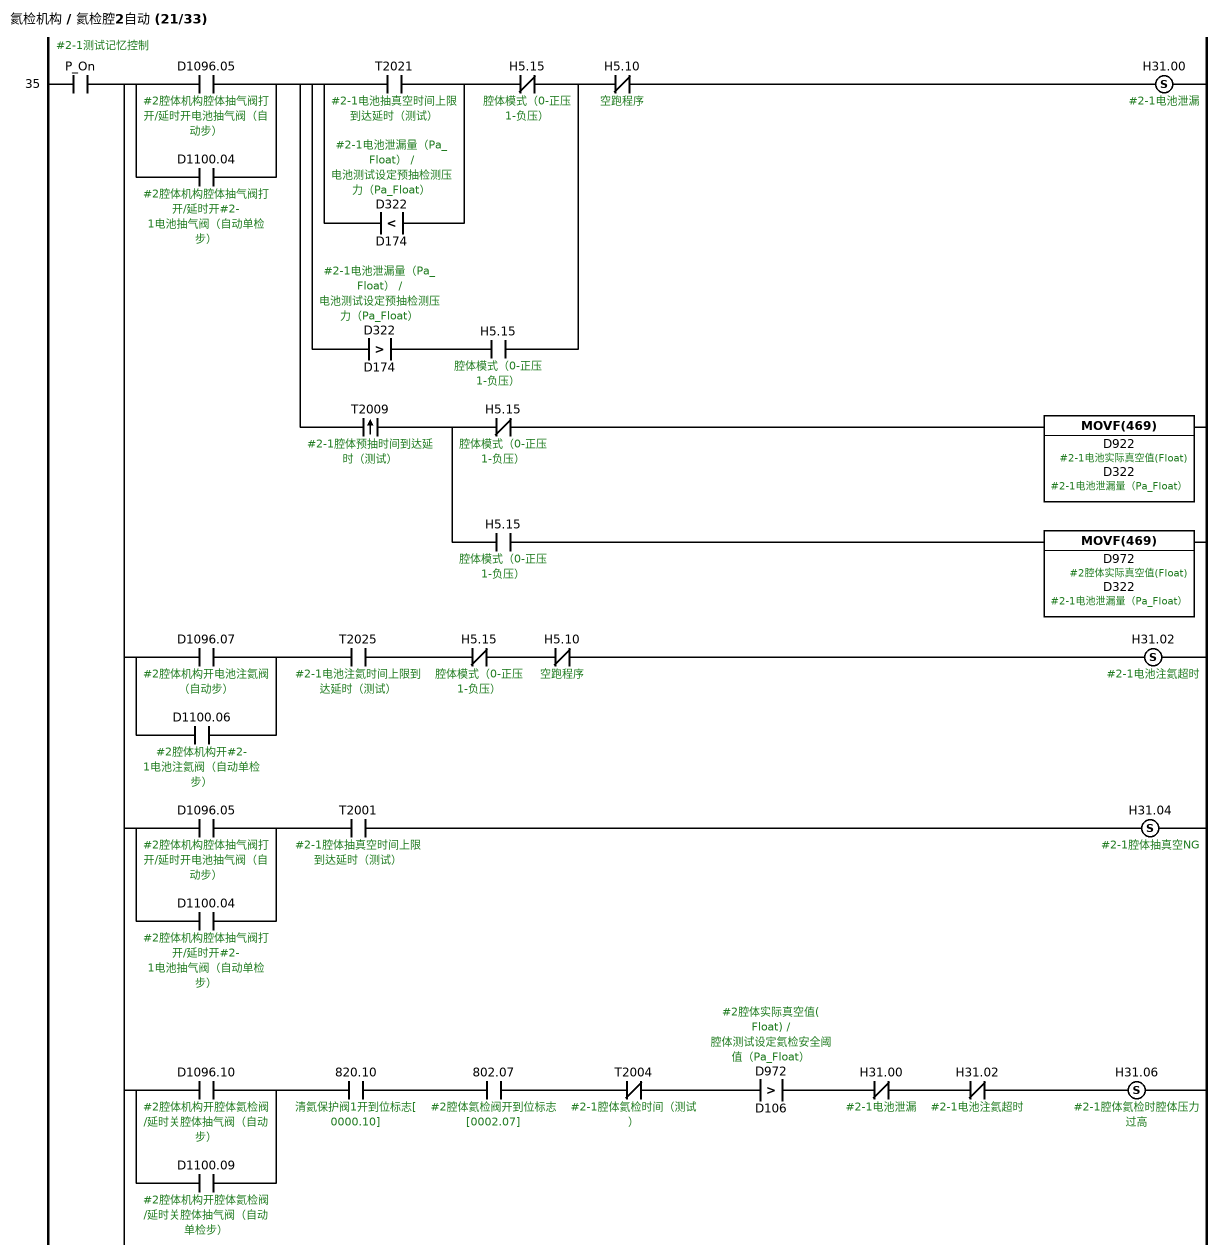

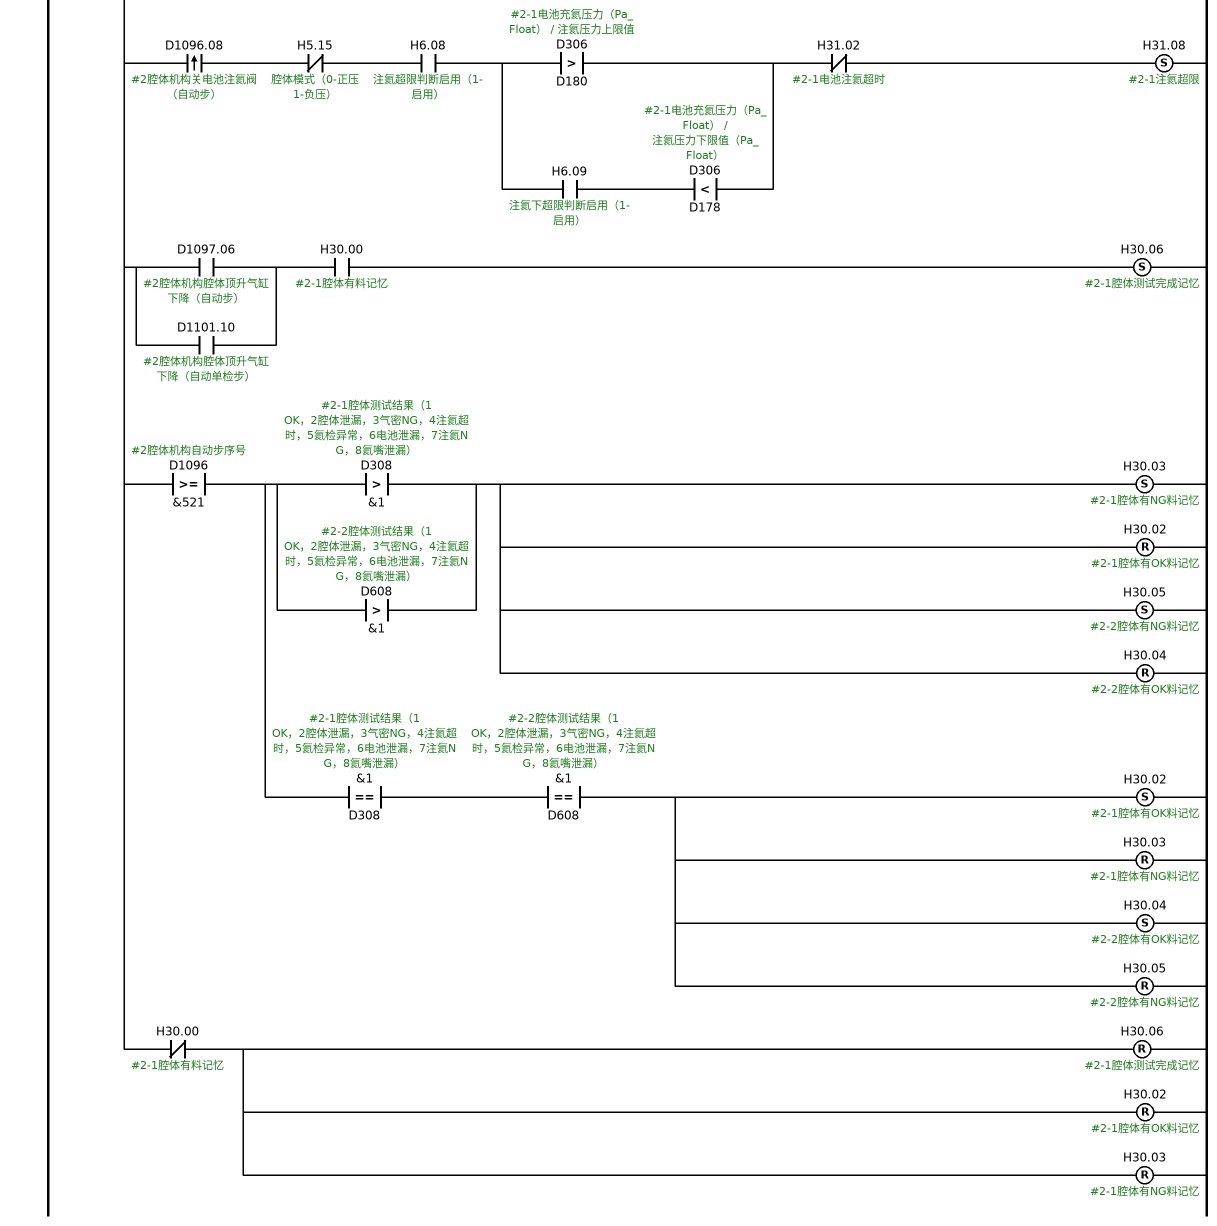
; rung 35: #2-1测试记忆控制
LD P_On
OUT TR0
LD D1096.05  ; #2腔体机构腔体抽气阀打开/延时开电池抽气阀（自动步）
OR D1100.04  ; #2腔体机构腔体抽气阀打开/延时开#2-1电池抽气阀（自动单检步）
ANDLD
OUT TR1
LD T2021  ; #2-1电池抽真空时间上限到达延时（测试）
OR<F(331) D322 D174  ; #2-1电池泄漏量（Pa_Float）, 电池测试设定预抽检测压力（Pa_Float）
ANDNOT H5.15  ; 腔体模式（0-正压 1-负压）
LD>F(333) D322 D174  ; #2-1电池泄漏量（Pa_Float）, 电池测试设定预抽检测压力（Pa_Float）
AND H5.15  ; 腔体模式（0-正压 1-负压）
ORLD
ANDLD
ANDNOT H5.10  ; 空跑程序
SET H31.00  ; #2-1电池泄漏
LD TR1
@AND T2009  ; #2-1腔体预抽时间到达延时（测试）
OUT TR1
ANDNOT H5.15  ; 腔体模式（0-正压 1-负压）
MOVF(469) D922 D322  ; #2-1电池实际真空值(Float), #2-1电池泄漏量（Pa_Float）
LD TR1
AND H5.15  ; 腔体模式（0-正压 1-负压）
MOVF(469) D972 D322  ; #2腔体实际真空值(Float), #2-1电池泄漏量（Pa_Float）
LD TR0
LD D1096.07  ; #2腔体机构开电池注氦阀（自动步）
OR D1100.06  ; #2腔体机构开#2-1电池注氦阀（自动单检步）
ANDLD
AND T2025  ; #2-1电池注氦时间上限到达延时（测试）
ANDNOT H5.15  ; 腔体模式（0-正压 1-负压）
ANDNOT H5.10  ; 空跑程序
SET H31.02  ; #2-1电池注氦超时
LD TR0
LD D1096.05  ; #2腔体机构腔体抽气阀打开/延时开电池抽气阀（自动步）
OR D1100.04  ; #2腔体机构腔体抽气阀打开/延时开#2-1电池抽气阀（自动单检步）
ANDLD
AND T2001  ; #2-1腔体抽真空时间上限到达延时（测试）
SET H31.04  ; #2-1腔体抽真空NG
LD TR0
LD D1096.10  ; #2腔体机构开腔体氦检阀/延时关腔体抽气阀（自动步）
OR D1100.09  ; #2腔体机构开腔体氦检阀/延时关腔体抽气阀（自动单检步）
ANDLD
AND 820.10  ; 清氦保护阀1开到位标志[0000.10]
AND 802.07  ; #2腔体氦检阀开到位标志[0002.07]
ANDNOT T2004  ; #2-1腔体氦检时间（测试）
AND>F(333) D972 D106  ; #2腔体实际真空值(Float), 腔体测试设定氦检安全阈值（Pa_Float）
ANDNOT H31.00  ; #2-1电池泄漏
ANDNOT H31.02  ; #2-1电池注氦超时
SET H31.06  ; #2-1腔体氦检时腔体压力过高
LD TR0
@AND D1096.08  ; #2腔体机构关电池注氦阀（自动步）
ANDNOT H5.15  ; 腔体模式（0-正压 1-负压）
AND H6.08  ; 注氦超限判断启用（1-启用）
LD>F(333) D306 D180  ; #2-1电池充氦压力（Pa_Float）, 注氦压力上限值
LD H6.09  ; 注氦下超限判断启用（1-启用）
AND<F(331) D306 D178  ; #2-1电池充氦压力（Pa_Float）, 注氦压力下限值（Pa_Float）
ORLD
ANDLD
ANDNOT H31.02  ; #2-1电池注氦超时
SET H31.08  ; #2-1注氦超限
LD TR0
LD D1097.06  ; #2腔体机构腔体顶升气缸下降（自动步）
OR D1101.10  ; #2腔体机构腔体顶升气缸下降（自动单检步）
ANDLD
AND H30.00  ; #2-1腔体有料记忆
SET H30.06  ; #2-1腔体测试完成记忆
LD TR0
AND>=L(326) D1096 &521  ; #2腔体机构自动步序号
OUT TR1
LD>(320) D308 &1  ; #2-1腔体测试结果（1 OK，2腔体泄漏，3气密NG，4注氦超时，5氦检异常，6电池泄漏，7注氦NG，8氦嘴泄漏）
OR>(320) D608 &1  ; #2-2腔体测试结果（1 OK，2腔体泄漏，3气密NG，4注氦超时，5氦检异常，6电池泄漏，7注氦NG，8氦嘴泄漏）
ANDLD
SET H30.03  ; #2-1腔体有NG料记忆
RSET H30.02  ; #2-1腔体有OK料记忆
SET H30.05  ; #2-2腔体有NG料记忆
RSET H30.04  ; #2-2腔体有OK料记忆
LD TR1
AND=(300) &1 D308  ; #2-1腔体测试结果（1 OK，2腔体泄漏，3气密NG，4注氦超时，5氦检异常，6电池泄漏，7注氦NG，8氦嘴泄漏）
AND=(300) &1 D608  ; #2-2腔体测试结果（1 OK，2腔体泄漏，3气密NG，4注氦超时，5氦检异常，6电池泄漏，7注氦NG，8氦嘴泄漏）
SET H30.02  ; #2-1腔体有OK料记忆
RSET H30.03  ; #2-1腔体有NG料记忆
SET H30.04  ; #2-2腔体有OK料记忆
RSET H30.05  ; #2-2腔体有NG料记忆
LD TR0
ANDNOT H30.00  ; #2-1腔体有料记忆
RSET H30.06  ; #2-1腔体测试完成记忆
RSET H30.02  ; #2-1腔体有OK料记忆
RSET H30.03  ; #2-1腔体有NG料记忆

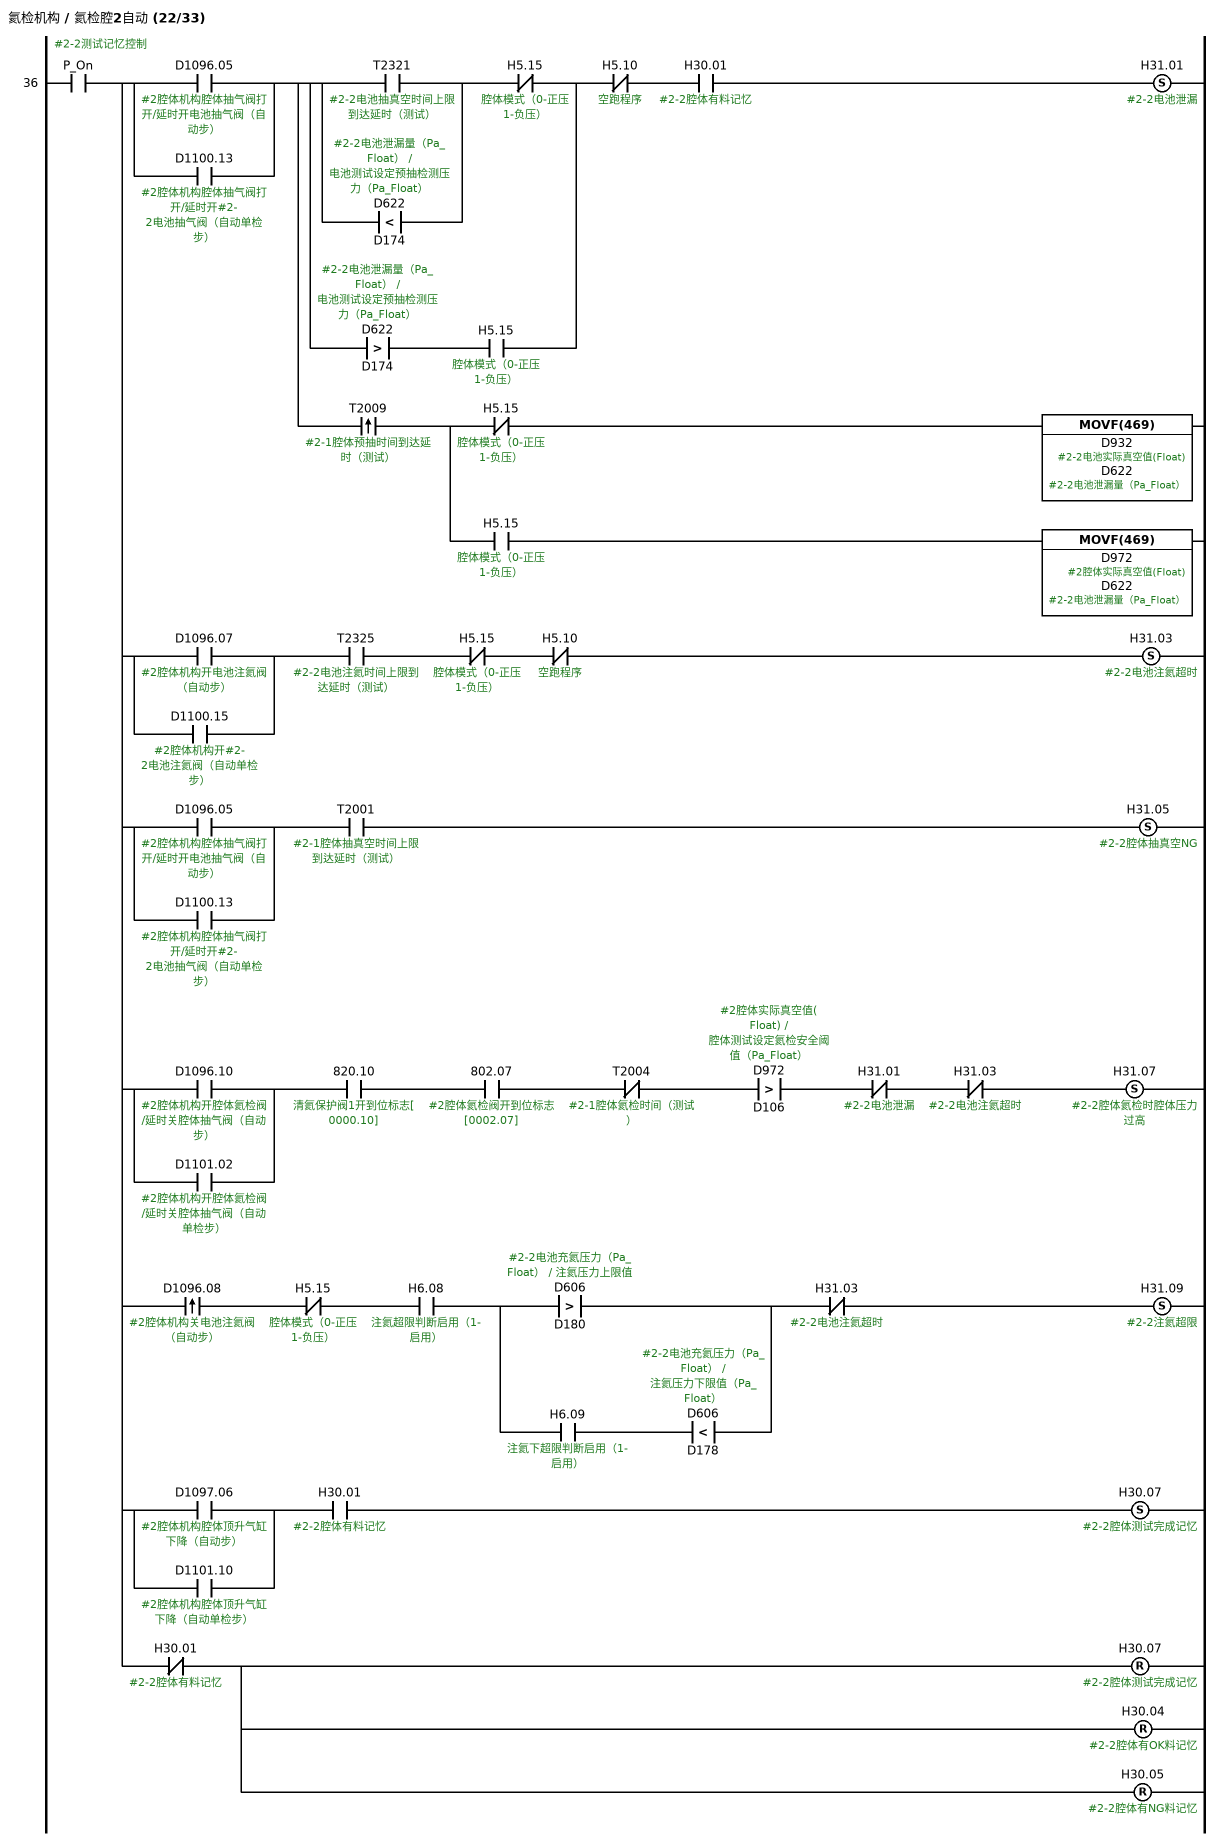
; rung 36: #2-2测试记忆控制
LD P_On
OUT TR0
LD D1096.05  ; #2腔体机构腔体抽气阀打开/延时开电池抽气阀（自动步）
OR D1100.13  ; #2腔体机构腔体抽气阀打开/延时开#2-2电池抽气阀（自动单检步）
ANDLD
OUT TR1
LD T2321  ; #2-2电池抽真空时间上限到达延时（测试）
OR<F(331) D622 D174  ; #2-2电池泄漏量（Pa_Float）, 电池测试设定预抽检测压力（Pa_Float）
ANDNOT H5.15  ; 腔体模式（0-正压 1-负压）
LD>F(333) D622 D174  ; #2-2电池泄漏量（Pa_Float）, 电池测试设定预抽检测压力（Pa_Float）
AND H5.15  ; 腔体模式（0-正压 1-负压）
ORLD
ANDLD
ANDNOT H5.10  ; 空跑程序
AND H30.01  ; #2-2腔体有料记忆
SET H31.01  ; #2-2电池泄漏
LD TR1
@AND T2009  ; #2-1腔体预抽时间到达延时（测试）
OUT TR1
ANDNOT H5.15  ; 腔体模式（0-正压 1-负压）
MOVF(469) D932 D622  ; #2-2电池实际真空值(Float), #2-2电池泄漏量（Pa_Float）
LD TR1
AND H5.15  ; 腔体模式（0-正压 1-负压）
MOVF(469) D972 D622  ; #2腔体实际真空值(Float), #2-2电池泄漏量（Pa_Float）
LD TR0
LD D1096.07  ; #2腔体机构开电池注氦阀（自动步）
OR D1100.15  ; #2腔体机构开#2-2电池注氦阀（自动单检步）
ANDLD
AND T2325  ; #2-2电池注氦时间上限到达延时（测试）
ANDNOT H5.15  ; 腔体模式（0-正压 1-负压）
ANDNOT H5.10  ; 空跑程序
SET H31.03  ; #2-2电池注氦超时
LD TR0
LD D1096.05  ; #2腔体机构腔体抽气阀打开/延时开电池抽气阀（自动步）
OR D1100.13  ; #2腔体机构腔体抽气阀打开/延时开#2-2电池抽气阀（自动单检步）
ANDLD
AND T2001  ; #2-1腔体抽真空时间上限到达延时（测试）
SET H31.05  ; #2-2腔体抽真空NG
LD TR0
LD D1096.10  ; #2腔体机构开腔体氦检阀/延时关腔体抽气阀（自动步）
OR D1101.02  ; #2腔体机构开腔体氦检阀/延时关腔体抽气阀（自动单检步）
ANDLD
AND 820.10  ; 清氦保护阀1开到位标志[0000.10]
AND 802.07  ; #2腔体氦检阀开到位标志[0002.07]
ANDNOT T2004  ; #2-1腔体氦检时间（测试）
AND>F(333) D972 D106  ; #2腔体实际真空值(Float), 腔体测试设定氦检安全阈值（Pa_Float）
ANDNOT H31.01  ; #2-2电池泄漏
ANDNOT H31.03  ; #2-2电池注氦超时
SET H31.07  ; #2-2腔体氦检时腔体压力过高
LD TR0
@AND D1096.08  ; #2腔体机构关电池注氦阀（自动步）
ANDNOT H5.15  ; 腔体模式（0-正压 1-负压）
AND H6.08  ; 注氦超限判断启用（1-启用）
LD>F(333) D606 D180  ; #2-2电池充氦压力（Pa_Float）, 注氦压力上限值
LD H6.09  ; 注氦下超限判断启用（1-启用）
AND<F(331) D606 D178  ; #2-2电池充氦压力（Pa_Float）, 注氦压力下限值（Pa_Float）
ORLD
ANDLD
ANDNOT H31.03  ; #2-2电池注氦超时
SET H31.09  ; #2-2注氦超限
LD TR0
LD D1097.06  ; #2腔体机构腔体顶升气缸下降（自动步）
OR D1101.10  ; #2腔体机构腔体顶升气缸下降（自动单检步）
ANDLD
AND H30.01  ; #2-2腔体有料记忆
SET H30.07  ; #2-2腔体测试完成记忆
LD TR0
ANDNOT H30.01  ; #2-2腔体有料记忆
RSET H30.07  ; #2-2腔体测试完成记忆
RSET H30.04  ; #2-2腔体有OK料记忆
RSET H30.05  ; #2-2腔体有NG料记忆

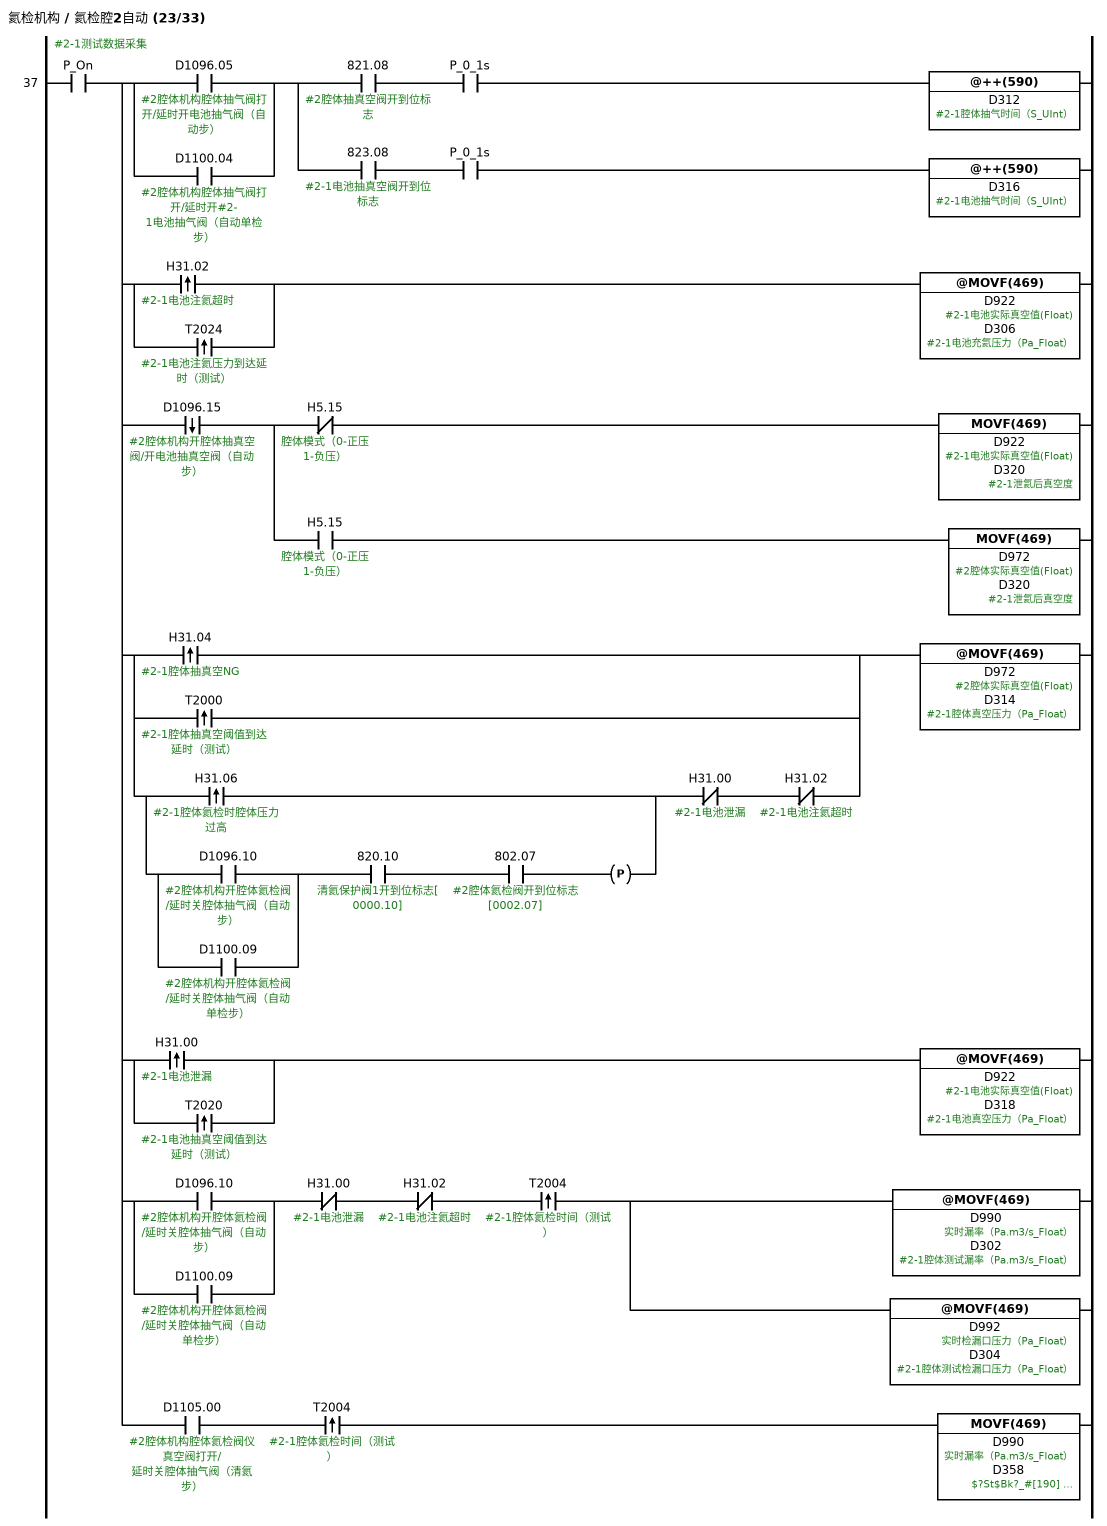
; rung 37: #2-1测试数据采集
LD P_On
OUT TR0
LD D1096.05  ; #2腔体机构腔体抽气阀打开/延时开电池抽气阀（自动步）
OR D1100.04  ; #2腔体机构腔体抽气阀打开/延时开#2-1电池抽气阀（自动单检步）
ANDLD
OUT TR1
AND 821.08  ; #2腔体抽真空阀开到位标志
AND P_0_1s
@++(590) D312  ; #2-1腔体抽气时间（S_UInt）
LD TR1
AND 823.08  ; #2-1电池抽真空阀开到位标志
AND P_0_1s
@++(590) D316  ; #2-1电池抽气时间（S_UInt）
LD TR0
@LD H31.02  ; #2-1电池注氦超时
@OR T2024  ; #2-1电池注氦压力到达延时（测试）
ANDLD
@MOVF(469) D922 D306  ; #2-1电池实际真空值(Float), #2-1电池充氦压力（Pa_Float）
LD TR0
%AND D1096.15  ; #2腔体机构开腔体抽真空阀/开电池抽真空阀（自动步）
OUT TR1
ANDNOT H5.15  ; 腔体模式（0-正压 1-负压）
MOVF(469) D922 D320  ; #2-1电池实际真空值(Float), #2-1泄氦后真空度
LD TR1
AND H5.15  ; 腔体模式（0-正压 1-负压）
MOVF(469) D972 D320  ; #2腔体实际真空值(Float), #2-1泄氦后真空度
LD TR0
@LD H31.04  ; #2-1腔体抽真空NG
@OR T2000  ; #2-1腔体抽真空阈值到达延时（测试）
@LD H31.06  ; #2-1腔体氦检时腔体压力过高
LD D1096.10  ; #2腔体机构开腔体氦检阀/延时关腔体抽气阀（自动步）
OR D1100.09  ; #2腔体机构开腔体氦检阀/延时关腔体抽气阀（自动单检步）
AND 820.10  ; 清氦保护阀1开到位标志[0000.10]
AND 802.07  ; #2腔体氦检阀开到位标志[0002.07]
UP(521)
ORLD
ANDNOT H31.00  ; #2-1电池泄漏
ANDNOT H31.02  ; #2-1电池注氦超时
ORLD
ANDLD
@MOVF(469) D972 D314  ; #2腔体实际真空值(Float), #2-1腔体真空压力（Pa_Float）
LD TR0
@LD H31.00  ; #2-1电池泄漏
@OR T2020  ; #2-1电池抽真空阈值到达延时（测试）
ANDLD
@MOVF(469) D922 D318  ; #2-1电池实际真空值(Float), #2-1电池真空压力（Pa_Float）
LD TR0
LD D1096.10  ; #2腔体机构开腔体氦检阀/延时关腔体抽气阀（自动步）
OR D1100.09  ; #2腔体机构开腔体氦检阀/延时关腔体抽气阀（自动单检步）
ANDLD
ANDNOT H31.00  ; #2-1电池泄漏
ANDNOT H31.02  ; #2-1电池注氦超时
@AND T2004  ; #2-1腔体氦检时间（测试）
@MOVF(469) D990 D302  ; 实时漏率（Pa.m3/s_Float）, #2-1腔体测试漏率（Pa.m3/s_Float）
@MOVF(469) D992 D304  ; 实时检漏口压力（Pa_Float）, #2-1腔体测试检漏口压力（Pa_Float）
LD TR0
AND D1105.00  ; #2腔体机构腔体氦检阀仪真空阀打开/延时关腔体抽气阀（清氦步）
@AND T2004  ; #2-1腔体氦检时间（测试）
MOVF(469) D990 D358  ; 实时漏率（Pa.m3/s_Float）, $?St$Bk?_#[190] / #2-1清氦泄漏率（清氦） / $?St$Bk?_#[190]

